C03633=1093.547,92.703,-61.297,175.902,17.512,152.547
C03634=1093.553,92.952,-61.315,175.903,17.513,152.547
C03635=1093.558,93.202,-61.333,175.906,17.514,152.547
C03636=1093.564,93.452,-61.351,175.908,17.515,152.547
C03637=1093.569,93.701,-61.369,175.911,17.516,152.546
C03638=1093.575,93.950,-61.386,175.913,17.517,152.546
C03639=1093.581,94.199,-61.405,175.915,17.518,152.546
C03640=1093.586,94.448,-61.423,175.918,17.519,152.546
C03641=1093.592,94.697,-61.441,175.920,17.520,152.545
C03642=1093.598,94.947,-61.459,175.923,17.521,152.545
C03643=1093.603,95.196,-61.476,175.925,17.522,152.545
C03644=1093.609,95.472,-61.497,175.927,17.523,152.545
C03645=1093.616,95.748,-61.516,175.930,17.524,152.544
C03646=1093.622,96.023,-61.536,175.933,17.525,152.544
C03647=1093.628,96.299,-61.557,175.935,17.526,152.544
C03648=1093.634,96.548,-61.575,175.938,17.528,152.544
C03649=1093.639,96.797,-61.592,175.940,17.529,152.543
C03650=1093.645,97.048,-61.611,175.942,17.530,152.543
C03651=1093.651,97.296,-61.629,175.944,17.531,152.543
C03652=1093.657,97.546,-61.647,175.947,17.532,152.543
C03653=1093.662,97.795,-61.664,175.950,17.533,152.542
C03654=1093.668,98.045,-61.683,175.952,17.534,152.542
C03655=1093.673,98.293,-61.701,175.954,17.535,152.542
C03656=1093.680,98.543,-61.719,175.956,17.535,152.542
C03657=1093.684,98.792,-61.737,175.959,17.537,152.541
C03658=1093.691,99.041,-61.756,175.961,17.537,152.541
C03659=1093.696,99.290,-61.773,175.964,17.538,152.541
C03660=1093.702,99.540,-61.791,175.966,17.540,152.541
C03661=1093.707,99.789,-61.810,175.968,17.540,152.540
C03662=1093.714,100.039,-61.828,175.971,17.541,152.540
C03663=1093.719,100.288,-61.846,175.973,17.542,152.540
C03664=1093.725,100.537,-61.865,175.976,17.543,152.540
C03665=1093.730,100.786,-61.883,175.978,17.545,152.539
C03666=1093.736,101.036,-61.901,175.980,17.545,152.539
C03667=1093.742,101.285,-61.919,175.983,17.546,152.539
C03668=1093.748,101.534,-61.937,175.985,17.547,152.538
C03669=1093.753,101.783,-61.956,175.988,17.548,152.538
C03670=1093.759,102.033,-61.974,175.990,17.549,152.538
C03671=1093.764,102.282,-61.993,175.992,17.550,152.538
C03672=1093.770,102.531,-62.011,175.995,17.551,152.537
C03673=1093.775,102.781,-62.029,175.998,17.552,152.537
C03674=1093.781,103.030,-62.048,176.000,17.553,152.537
C03675=1093.786,103.279,-62.066,176.002,17.554,152.537
C03676=1093.792,103.528,-62.085,176.004,17.555,152.536
C03677=1093.797,103.778,-62.103,176.007,17.556,152.536
C03678=1093.804,104.027,-62.121,176.010,17.557,152.536
C03679=1093.808,104.276,-62.140,176.012,17.558,152.536
C03680=1093.815,104.525,-62.158,176.014,17.559,152.535
C03681=1093.820,104.775,-62.176,176.016,17.559,152.535
C03682=1093.826,105.024,-62.195,176.019,17.560,152.535
C03683=1093.831,105.273,-62.213,176.022,17.562,152.534
C03684=1093.837,105.522,-62.232,176.024,17.562,152.534
C03685=1093.842,105.771,-62.251,176.027,17.563,152.534
C03686=1093.848,106.021,-62.269,176.029,17.565,152.534
C03687=1093.854,106.269,-62.288,176.031,17.565,152.533
C03688=1093.859,106.519,-62.306,176.034,17.566,152.533
C03689=1093.865,106.769,-62.325,176.036,17.567,152.533
C03690=1093.870,107.017,-62.344,176.039,17.568,152.532
C03691=1093.877,107.267,-62.362,176.041,17.569,152.532
C03692=1093.882,107.516,-62.380,176.043,17.570,152.532
C03693=1093.887,107.766,-62.399,176.046,17.571,152.532
C03694=1093.893,108.015,-62.418,176.049,17.572,152.531
C03695=1093.899,108.264,-62.436,176.051,17.573,152.531
C03696=1093.905,108.513,-62.454,176.054,17.573,152.531
C03697=1093.910,108.762,-62.473,176.056,17.574,152.530
C03698=1093.915,109.012,-62.492,176.058,17.575,152.530
C03699=1093.922,109.261,-62.510,176.061,17.576,152.530
C03700=1093.927,109.510,-62.529,176.063,17.577,152.530
C03701=1093.933,109.759,-62.548,176.066,17.578,152.529
C03702=1093.939,110.009,-62.567,176.069,17.579,152.529
C03703=1093.944,110.258,-62.585,176.071,17.580,152.529
C03704=1093.950,110.507,-62.604,176.073,17.581,152.528
C03705=1093.956,110.757,-62.623,176.075,17.581,152.528
C03706=1093.962,111.005,-62.642,176.078,17.582,152.528
C03707=1093.967,111.255,-62.660,176.081,17.583,152.528
C03708=1093.973,111.531,-62.681,176.084,17.584,152.527
C03709=1093.979,111.806,-62.702,176.087,17.585,152.527
C03710=1093.985,112.082,-62.723,176.089,17.586,152.527
C03711=1093.992,112.359,-62.744,176.092,17.587,152.526
C03712=1093.997,112.607,-62.762,176.094,17.588,152.526
C03713=1094.003,112.856,-62.781,176.097,17.589,152.526
C03714=1094.009,113.106,-62.801,176.099,17.589,152.525
C03715=1094.014,113.355,-62.819,176.102,17.590,152.525
C03716=1094.020,113.604,-62.837,176.105,17.592,152.525
C03717=1094.026,113.854,-62.857,176.107,17.592,152.524
C03718=1094.031,114.103,-62.876,176.109,17.593,152.524
C03719=1094.036,114.352,-62.895,176.112,17.594,152.524
C03720=1094.043,114.601,-62.913,176.114,17.595,152.524
C03721=1094.049,114.850,-62.933,176.117,17.595,152.523
C03722=1094.054,115.099,-62.952,176.120,17.597,152.523
C03723=1094.059,115.349,-62.971,176.122,17.597,152.523
C03724=1094.065,115.598,-62.990,176.124,17.598,152.522
C03725=1094.070,115.847,-63.009,176.127,17.599,152.522
C03726=1094.076,116.096,-63.028,176.129,17.600,152.522
C03727=1094.081,116.346,-63.047,176.132,17.601,152.521
C03728=1094.086,116.595,-63.066,176.134,17.602,152.521
C03729=1094.092,116.844,-63.085,176.137,17.602,152.521
C03730=1094.098,117.094,-63.104,176.140,17.604,152.520
C03731=1094.103,117.343,-63.123,176.142,17.604,152.520
C03732=1094.108,117.592,-63.142,176.145,17.605,152.520
C03733=1094.114,117.842,-63.161,176.147,17.606,152.520
C03734=1094.119,118.090,-63.180,176.149,17.607,152.519
C03735=1094.126,118.339,-63.199,176.152,17.607,152.519
C03736=1094.132,118.588,-63.219,176.155,17.609,152.519
C03737=1094.137,118.838,-63.238,176.157,17.609,152.518
C03738=1094.142,119.086,-63.257,176.160,17.610,152.518
C03739=1094.148,119.336,-63.276,176.163,17.611,152.518
C03740=1094.154,119.585,-63.295,176.165,17.611,152.517
C03741=1094.159,119.835,-63.315,176.167,17.613,152.517
C03742=1094.165,120.083,-63.334,176.170,17.614,152.517
C03743=1094.170,120.333,-63.353,176.172,17.614,152.516
C03744=1094.176,120.582,-63.372,176.175,17.615,152.516
C03745=1094.182,120.832,-63.391,176.178,17.616,152.516
C03746=1094.187,121.080,-63.410,176.181,17.617,152.515
C03747=1094.193,121.329,-63.430,176.183,17.617,152.515
C03748=1094.198,121.579,-63.449,176.186,17.618,152.515
C03749=1094.204,121.828,-63.469,176.188,17.620,152.515
C03750=1094.210,122.078,-63.488,176.191,17.620,152.514
C03751=1094.215,122.326,-63.507,176.193,17.621,152.514
C03752=1094.220,122.575,-63.527,176.196,17.622,152.513
C03753=1094.226,122.825,-63.547,176.198,17.622,152.513
C03754=1094.231,123.074,-63.566,176.201,17.623,152.513
C03755=1094.237,123.324,-63.585,176.204,17.624,152.512
C03756=1094.242,123.572,-63.604,176.206,17.624,152.512
C03757=1094.248,123.821,-63.624,176.209,17.626,152.512
C03758=1094.254,124.071,-63.643,176.212,17.626,152.511
C03759=1094.260,124.320,-63.662,176.214,17.627,152.511
C03760=1094.266,124.569,-63.682,176.217,17.628,152.511
C03761=1094.271,124.818,-63.702,176.220,17.628,152.510
C03762=1094.277,125.068,-63.721,176.222,17.629,152.510
C03763=1094.282,125.316,-63.740,176.225,17.630,152.510
C03764=1094.288,125.565,-63.760,176.227,17.631,152.509
C03765=1094.294,125.815,-63.779,176.229,17.631,152.509
C03766=1094.299,126.064,-63.798,176.232,17.632,152.509
C03767=1094.305,126.313,-63.819,176.235,17.633,152.508
C03768=1094.310,126.563,-63.838,176.238,17.634,152.508
C03769=1094.316,126.812,-63.858,176.240,17.634,152.508
C03770=1094.322,127.061,-63.877,176.243,17.635,152.507
C03771=1094.328,127.310,-63.896,176.246,17.636,152.507
C03772=1094.334,127.586,-63.918,176.249,17.637,152.506
C03773=1094.340,127.862,-63.940,176.252,17.638,152.506
C03774=1094.347,128.138,-63.961,176.255,17.639,152.506
C03775=1094.353,128.413,-63.983,176.258,17.639,152.505
C03776=1094.358,128.663,-64.003,176.260,17.639,152.505
C03777=1094.364,128.912,-64.023,176.263,17.641,152.505
C03778=1094.370,129.161,-64.042,176.266,17.641,152.504
C03779=1094.376,129.410,-64.062,176.268,17.642,152.504
C03780=1094.382,129.659,-64.081,176.271,17.642,152.503
C03781=1094.388,129.908,-64.101,176.274,17.643,152.503
C03782=1094.393,130.158,-64.121,176.276,17.644,152.503
C03783=1094.398,130.407,-64.141,176.279,17.644,152.502
C03784=1094.404,130.656,-64.160,176.282,17.645,152.502
C03785=1094.410,130.905,-64.180,176.284,17.646,152.502
C03786=1094.416,131.154,-64.200,176.287,17.646,152.501
C03787=1094.422,131.403,-64.220,176.290,17.647,152.501
C03788=1094.427,131.653,-64.239,176.293,17.648,152.500
C03789=1094.433,131.902,-64.259,176.294,17.649,152.500
C03790=1094.439,132.151,-64.279,176.297,17.649,152.500
C03791=1094.444,132.400,-64.299,176.300,17.650,152.499
C03792=1094.450,132.649,-64.319,176.303,17.650,152.499
C03793=1094.455,132.898,-64.338,176.305,17.651,152.499
C03794=1094.461,133.147,-64.358,176.308,17.652,152.498
C03795=1094.466,133.396,-64.379,176.311,17.653,152.498
C03796=1094.472,133.645,-64.398,176.313,17.653,152.498
C03797=1094.477,133.894,-64.418,176.316,17.654,152.497
C03798=1094.483,134.144,-64.438,176.319,17.655,152.497
C03799=1094.489,134.393,-64.458,176.322,17.656,152.496
C03800=1094.494,134.642,-64.478,176.324,17.656,152.496
C03801=1094.500,134.891,-64.498,176.327,17.657,152.496
C03802=1094.505,135.140,-64.518,176.330,17.658,152.495
C03803=1094.511,135.389,-64.538,176.332,17.658,152.495
C03804=1094.517,135.638,-64.558,176.335,17.659,152.495
C03805=1094.522,135.888,-64.578,176.338,17.659,152.494
C03806=1094.528,136.137,-64.598,176.341,17.661,152.494
C03807=1094.534,136.386,-64.619,176.343,17.661,152.493
C03808=1094.540,136.635,-64.638,176.346,17.661,152.493
C03809=1094.545,136.885,-64.658,176.349,17.662,152.493
C03810=1094.551,137.134,-64.678,176.352,17.663,152.492
C03811=1094.557,137.383,-64.698,176.354,17.663,152.492
C03812=1094.562,137.632,-64.719,176.357,17.664,152.492
C03813=1094.568,137.880,-64.739,176.360,17.665,152.491
C03814=1094.573,138.130,-64.759,176.362,17.665,152.491
C03815=1094.579,138.379,-64.779,176.365,17.666,152.490
C03816=1094.584,138.628,-64.799,176.368,17.667,152.490
C03817=1094.590,138.877,-64.819,176.371,17.667,152.490
C03818=1094.595,139.126,-64.840,176.373,17.668,152.489
C03819=1094.601,139.375,-64.860,176.376,17.668,152.489
C03820=1094.606,139.625,-64.879,176.379,17.669,152.488
C03821=1094.613,139.874,-64.900,176.382,17.670,152.488
C03822=1094.618,140.123,-64.920,176.384,17.670,152.488
C03823=1094.624,140.372,-64.940,176.387,17.671,152.487
C03824=1094.629,140.621,-64.961,176.390,17.672,152.487
C03825=1094.635,140.870,-64.981,176.393,17.673,152.486
C03826=1094.641,141.119,-65.001,176.395,17.673,152.486
C03827=1094.646,141.368,-65.022,176.398,17.674,152.486
C03828=1094.652,141.617,-65.042,176.401,17.674,152.485
C03829=1094.657,141.866,-65.062,176.404,17.675,152.485
C03830=1094.662,142.115,-65.083,176.406,17.675,152.484
C03831=1094.669,142.365,-65.103,176.409,17.676,152.484
C03832=1094.674,142.614,-65.124,176.412,17.677,152.484
C03833=1094.679,142.863,-65.144,176.415,17.677,152.483
C03834=1094.685,143.112,-65.164,176.418,17.678,152.483
C03835=1094.691,143.361,-65.185,176.420,17.679,152.482
C03836=1094.697,143.637,-65.207,176.424,17.679,152.482
C03837=1094.703,143.913,-65.230,176.427,17.680,152.482
C03838=1094.709,144.189,-65.253,176.430,17.681,152.481
C03839=1094.715,144.464,-65.275,176.432,17.681,152.481
C03840=1094.721,144.713,-65.295,176.435,17.682,152.480
C03841=1094.726,144.962,-65.316,176.438,17.683,152.480
C03842=1094.732,145.212,-65.337,176.441,17.683,152.479
C03843=1094.739,145.460,-65.357,176.444,17.684,152.479
C03844=1094.744,145.709,-65.378,176.447,17.684,152.479
C03845=1094.749,145.958,-65.399,176.450,17.685,152.478
C03846=1094.754,146.208,-65.419,176.453,17.685,152.478
C03847=1094.761,146.457,-65.439,176.455,17.686,152.477
C03848=1094.766,146.706,-65.460,176.458,17.686,152.477
C03849=1094.771,146.955,-65.481,176.461,17.687,152.476
C03850=1094.778,147.203,-65.501,176.464,17.688,152.476
C03851=1094.784,147.453,-65.522,176.467,17.689,152.476
C03852=1094.789,147.702,-65.543,176.469,17.689,152.475
C03853=1094.794,147.952,-65.563,176.472,17.689,152.475
C03854=1094.800,148.200,-65.583,176.475,17.690,152.474
C03855=1094.806,148.449,-65.604,176.478,17.690,152.474
C03856=1094.812,148.699,-65.625,176.481,17.691,152.473
C03857=1094.817,148.948,-65.646,176.484,17.691,152.473
C03858=1094.822,149.197,-65.666,176.487,17.692,152.473
C03859=1094.828,149.445,-65.688,176.490,17.693,152.472
C03860=1094.834,149.695,-65.708,176.493,17.694,152.472
C03861=1094.839,149.944,-65.729,176.495,17.694,152.471
C03862=1094.845,150.193,-65.750,176.498,17.694,152.471
C03863=1094.850,150.442,-65.770,176.501,17.695,152.471
C03864=1094.856,150.692,-65.791,176.504,17.695,152.470
C03865=1094.862,150.940,-65.813,176.506,17.696,152.470
C03866=1094.867,151.189,-65.833,176.509,17.696,152.469
C03867=1094.872,151.438,-65.854,176.512,17.697,152.469
C03868=1094.878,151.687,-65.875,176.515,17.698,152.468
C03869=1094.884,151.936,-65.895,176.518,17.699,152.468
C03870=1094.890,152.185,-65.916,176.520,17.698,152.467
C03871=1094.896,152.435,-65.938,176.523,17.699,152.467
C03872=1094.901,152.684,-65.958,176.526,17.700,152.467
C03873=1094.907,152.932,-65.979,176.529,17.701,152.466
C03874=1094.912,153.181,-66.000,176.532,17.701,152.466
C03875=1094.918,153.431,-66.021,176.535,17.701,152.465
C03876=1094.923,153.680,-66.042,176.538,17.702,152.465
C03877=1094.929,153.929,-66.063,176.541,17.702,152.464
C03878=1094.935,154.178,-66.084,176.544,17.703,152.464
C03879=1094.940,154.427,-66.105,176.547,17.704,152.463
C03880=1094.946,154.676,-66.126,176.549,17.704,152.463
C03881=1094.951,154.925,-66.147,176.552,17.704,152.463
C03882=1094.957,155.174,-66.168,176.555,17.705,152.462
C03883=1094.962,155.423,-66.189,176.559,17.705,152.462
C03884=1094.968,155.672,-66.210,176.561,17.706,152.461
C03885=1094.974,155.921,-66.231,176.564,17.706,152.461
C03886=1094.979,156.170,-66.252,176.567,17.707,152.460
C03887=1094.985,156.420,-66.273,176.570,17.707,152.460
C03888=1094.991,156.668,-66.294,176.573,17.708,152.460
C03889=1094.997,156.917,-66.316,176.576,17.709,152.459
C03890=1095.002,157.167,-66.337,176.578,17.709,152.459
C03891=1095.008,157.415,-66.358,176.581,17.709,152.458
C03892=1095.013,157.665,-66.379,176.584,17.710,152.458
C03893=1095.018,157.914,-66.401,176.587,17.711,152.457
C03894=1095.024,158.162,-66.422,176.591,17.711,152.457
C03895=1095.030,158.412,-66.443,176.594,17.712,152.456
C03896=1095.035,158.661,-66.464,176.596,17.712,152.456
C03897=1095.041,158.910,-66.486,176.599,17.712,152.455
C03898=1095.047,159.159,-66.506,176.602,17.713,152.455
C03899=1095.052,159.407,-66.528,176.605,17.714,152.455
C03900=1095.058,159.683,-66.552,176.608,17.714,152.454
C03901=1095.065,159.958,-66.575,176.611,17.714,152.453
C03902=1095.071,160.234,-66.599,176.614,17.715,152.453
C03903=1095.077,160.509,-66.622,176.618,17.715,152.453
C03904=1095.083,160.759,-66.643,176.621,17.716,152.452
C03905=1095.088,161.008,-66.665,176.624,17.716,152.452
C03906=1095.094,161.256,-66.686,176.627,17.717,152.451
C03907=1095.099,161.506,-66.708,176.630,17.717,152.451
C03908=1095.105,161.754,-66.729,176.632,17.718,152.450
C03909=1095.111,162.004,-66.750,176.635,17.718,152.450
C03910=1095.116,162.253,-66.772,176.639,17.719,152.449
C03911=1095.121,162.501,-66.793,176.642,17.719,152.449
C03912=1095.127,162.751,-66.815,176.645,17.720,152.448
C03913=1095.132,162.999,-66.837,176.648,17.720,152.448
C03914=1095.138,163.249,-66.858,176.651,17.721,152.447
C03915=1095.143,163.498,-66.880,176.653,17.721,152.447
C03916=1095.149,163.747,-66.901,176.656,17.722,152.446
C03917=1095.155,163.996,-66.923,176.659,17.722,152.446
C03918=1095.159,164.245,-66.945,176.662,17.723,152.446
C03919=1095.166,164.494,-66.966,176.665,17.723,152.445
C03920=1095.170,164.743,-66.988,176.668,17.724,152.445
C03921=1095.176,164.992,-67.009,176.671,17.724,152.444
C03922=1095.181,165.241,-67.031,176.674,17.725,152.444
C03923=1095.187,165.490,-67.052,176.677,17.725,152.443
C03924=1095.193,165.739,-67.074,176.680,17.726,152.443
C03925=1095.198,165.988,-67.096,176.683,17.726,152.442
C03926=1095.204,166.237,-67.117,176.686,17.727,152.442
C03927=1095.209,166.486,-67.139,176.689,17.728,152.441
C03928=1095.215,166.735,-67.161,176.691,17.728,152.441
C03929=1095.220,166.984,-67.183,176.695,17.728,152.440
C03930=1095.226,167.233,-67.204,176.698,17.729,152.440
C03931=1095.231,167.482,-67.226,176.701,17.729,152.439
C03932=1095.237,167.731,-67.248,176.704,17.730,152.439
C03933=1095.242,167.980,-67.270,176.707,17.730,152.439
C03934=1095.248,168.229,-67.291,176.710,17.731,152.438
C03935=1095.253,168.478,-67.313,176.713,17.731,152.438
C03936=1095.259,168.727,-67.335,176.716,17.731,152.437
C03937=1095.264,168.975,-67.357,176.719,17.732,152.437
C03938=1095.270,169.224,-67.379,176.722,17.732,152.436
C03939=1095.276,169.474,-67.401,176.725,17.733,152.436
C03940=1095.281,169.723,-67.422,176.728,17.733,152.435
C03941=1095.287,169.972,-67.445,176.731,17.734,152.435
C03942=1095.292,170.221,-67.466,176.734,17.734,152.434
C03943=1095.297,170.470,-67.488,176.737,17.734,152.434
C03944=1095.303,170.719,-67.509,176.740,17.735,152.433
C03945=1095.309,170.967,-67.532,176.743,17.735,152.433
C03946=1095.315,171.217,-67.554,176.746,17.735,152.432
C03947=1095.320,171.465,-67.576,176.749,17.736,152.432
C03948=1095.326,171.715,-67.598,176.752,17.737,152.431
C03949=1095.331,171.963,-67.619,176.755,17.737,152.431
C03950=1095.336,172.212,-67.642,176.759,17.738,152.430
C03951=1095.343,172.462,-67.664,176.761,17.737,152.430
C03952=1095.347,172.710,-67.686,176.764,17.738,152.429
C03953=1095.354,172.960,-67.707,176.767,17.738,152.429
C03954=1095.359,173.208,-67.730,176.770,17.739,152.428
C03955=1095.365,173.457,-67.752,176.774,17.739,152.428
C03956=1095.370,173.707,-67.774,176.777,17.740,152.427
C03957=1095.375,173.955,-67.796,176.780,17.740,152.427
C03958=1095.382,174.204,-67.818,176.783,17.741,152.426
C03959=1095.387,174.453,-67.840,176.786,17.740,152.426
C03960=1095.393,174.702,-67.862,176.789,17.741,152.425
C03961=1095.398,174.951,-67.885,176.792,17.742,152.425
C03962=1095.404,175.200,-67.907,176.795,17.742,152.424
C03963=1095.410,175.448,-67.929,176.798,17.742,152.424
C03964=1095.416,175.724,-67.953,176.802,17.742,152.423
C03965=1095.422,175.999,-67.978,176.805,17.743,152.423
C03966=1095.428,176.274,-68.002,176.809,17.744,152.422
C03967=1095.434,176.549,-68.027,176.812,17.744,152.421
C03968=1095.440,176.798,-68.049,176.815,17.745,152.421
C03969=1095.446,177.047,-68.072,176.818,17.745,152.420
C03970=1095.451,177.297,-68.094,176.822,17.745,152.420
C03971=1095.457,177.544,-68.116,176.824,17.745,152.419
C03972=1095.463,177.794,-68.138,176.827,17.745,152.419
C03973=1095.468,178.043,-68.161,176.830,17.746,152.418
C03974=1095.474,178.292,-68.183,176.834,17.746,152.418
C03975=1095.480,178.540,-68.205,176.837,17.747,152.417
C03976=1095.485,178.790,-68.227,176.840,17.747,152.417
C03977=1095.491,179.038,-68.250,176.843,17.747,152.416
C03978=1095.497,179.288,-68.272,176.846,17.748,152.416
C03979=1095.503,179.537,-68.295,176.850,17.748,152.415
C03980=1095.508,179.785,-68.316,176.853,17.749,152.415
C03981=1095.514,180.034,-68.339,176.855,17.748,152.414
C03982=1095.520,180.283,-68.362,176.858,17.749,152.414
C03983=1095.525,180.533,-68.384,176.862,17.749,152.413
C03984=1095.532,180.781,-68.407,176.865,17.749,152.412
C03985=1095.536,181.030,-68.429,176.868,17.750,152.412
C03986=1095.542,181.279,-68.451,176.871,17.750,152.412
C03987=1095.548,181.528,-68.474,176.874,17.751,152.411
C03988=1095.554,181.777,-68.496,176.878,17.751,152.410
C03989=1095.560,182.026,-68.519,176.881,17.751,152.410
C03990=1095.565,182.275,-68.542,176.884,17.751,152.409
C03991=1095.570,182.524,-68.564,176.887,17.752,152.409
C03992=1095.577,182.772,-68.586,176.891,17.752,152.408
C03993=1095.582,183.021,-68.609,176.893,17.752,152.408
C03994=1095.588,183.271,-68.631,176.896,17.752,152.407
C03995=1095.594,183.520,-68.654,176.900,17.752,152.407
C03996=1095.600,183.768,-68.677,176.903,17.753,152.406
C03997=1095.606,184.017,-68.700,176.906,17.753,152.405
C03998=1095.611,184.267,-68.722,176.909,17.753,152.405
C03999=1095.617,184.515,-68.745,176.913,17.754,152.404
C04000=1095.622,184.764,-68.767,176.916,17.754,152.404
C04001=1095.629,185.012,-68.790,176.919,17.754,152.403
C04002=1095.634,185.261,-68.813,176.922,17.755,152.403
C04003=1095.640,185.511,-68.835,176.925,17.755,152.402
C04004=1095.645,185.760,-68.858,176.929,17.756,152.402
C04005=1095.650,186.009,-68.881,176.932,17.756,152.401
C04006=1095.656,186.257,-68.904,176.935,17.756,152.401
C04007=1095.661,186.506,-68.927,176.938,17.757,152.400
C04008=1095.667,186.755,-68.950,176.941,17.757,152.400
C04009=1095.672,187.004,-68.972,176.944,17.757,152.399
C04010=1095.678,187.253,-68.995,176.947,17.757,152.399
C04011=1095.684,187.502,-69.018,176.950,17.758,152.398
C04012=1095.689,187.750,-69.040,176.954,17.758,152.397
C04013=1095.694,187.999,-69.064,176.957,17.758,152.397
C04014=1095.700,188.248,-69.087,176.960,17.759,152.396
C04015=1095.706,188.497,-69.110,176.963,17.759,152.396
C04016=1095.711,188.746,-69.133,176.966,17.760,152.395
C04017=1095.717,188.995,-69.156,176.970,17.760,152.395
C04018=1095.723,189.244,-69.179,176.973,17.760,152.394
C04019=1095.728,189.492,-69.201,176.976,17.761,152.394
C04020=1095.733,189.741,-69.225,176.979,17.761,152.393
C04021=1095.739,189.990,-69.248,176.983,17.761,152.393
C04022=1095.744,190.239,-69.271,176.986,17.762,152.392
C04023=1095.750,190.488,-69.294,176.989,17.762,152.392
C04024=1095.756,190.737,-69.317,176.992,17.762,152.391
C04025=1095.761,190.986,-69.340,176.996,17.763,152.390
C04026=1095.766,191.235,-69.363,176.999,17.763,152.390
C04027=1095.772,191.484,-69.386,177.002,17.763,152.389
C04028=1095.778,191.758,-69.411,177.005,17.763,152.389
C04029=1095.784,192.034,-69.437,177.009,17.764,152.388
C04030=1095.791,192.308,-69.462,177.013,17.765,152.388
C04031=1095.796,192.583,-69.488,177.016,17.765,152.387
C04032=1095.802,192.832,-69.511,177.019,17.765,152.386
C04033=1095.808,193.081,-69.534,177.023,17.765,152.386
C04034=1095.813,193.329,-69.557,177.026,17.765,152.385
C04035=1095.819,193.578,-69.581,177.029,17.766,152.385
C04036=1095.824,193.827,-69.604,177.032,17.766,152.384
C04037=1095.830,194.076,-69.627,177.036,17.766,152.384
C04038=1095.836,194.325,-69.650,177.039,17.767,152.383
C04039=1095.842,194.574,-69.673,177.042,17.767,152.382
C04040=1095.847,194.822,-69.697,177.045,17.767,152.382
C04041=1095.853,195.071,-69.720,177.049,17.768,152.381
C04042=1095.858,195.320,-69.743,177.052,17.768,152.381
C04043=1095.863,195.569,-69.767,177.055,17.768,152.380
C04044=1095.869,195.818,-69.791,177.058,17.769,152.380
C04045=1095.875,196.066,-69.813,177.062,17.769,152.379
C04046=1095.881,196.315,-69.836,177.065,17.769,152.378
C04047=1095.886,196.564,-69.861,177.068,17.769,152.378
C04048=1095.892,196.813,-69.884,177.072,17.769,152.377
C04049=1095.898,197.062,-69.907,177.075,17.770,152.377
C04050=1095.904,197.311,-69.931,177.078,17.770,152.376
C04051=1095.909,197.560,-69.954,177.081,17.770,152.376
C04052=1095.915,197.809,-69.977,177.085,17.771,152.375
C04053=1095.920,198.057,-70.001,177.088,17.771,152.375
C04054=1095.926,198.306,-70.024,177.091,17.771,152.374
C04055=1095.932,198.555,-70.047,177.095,17.771,152.373
C04056=1095.937,198.804,-70.072,177.098,17.772,152.373
C04057=1095.943,199.053,-70.094,177.101,17.772,152.372
C04058=1095.949,199.301,-70.118,177.104,17.772,152.372
C04059=1095.954,199.550,-70.142,177.108,17.772,152.371
C04060=1095.960,199.799,-70.166,177.111,17.772,152.370
C04061=1095.965,200.048,-70.189,177.114,17.773,152.370
C04062=1095.972,200.297,-70.213,177.118,17.773,152.369
C04063=1095.977,200.545,-70.236,177.121,17.773,152.369
C04064=1095.983,200.794,-70.260,177.124,17.773,152.368
C04065=1095.988,201.043,-70.283,177.128,17.774,152.368
C04066=1095.995,201.292,-70.307,177.131,17.774,152.367
C04067=1096.000,201.541,-70.331,177.134,17.774,152.366
C04068=1096.006,201.789,-70.354,177.138,17.774,152.366
C04069=1096.011,202.039,-70.378,177.141,17.774,152.365
C04070=1096.017,202.287,-70.401,177.144,17.775,152.365
C04071=1096.023,202.537,-70.425,177.147,17.775,152.364
C04072=1096.029,202.785,-70.449,177.151,17.775,152.363
C04073=1096.034,203.034,-70.473,177.154,17.775,152.363
C04074=1096.040,203.283,-70.496,177.157,17.776,152.362
C04075=1096.045,203.531,-70.520,177.161,17.776,152.362
C04076=1096.051,203.780,-70.543,177.164,17.776,152.361
C04077=1096.057,204.029,-70.568,177.167,17.777,152.361
C04078=1096.063,204.278,-70.592,177.171,17.776,152.360
C04079=1096.068,204.527,-70.615,177.174,17.777,152.359
C04080=1096.073,204.775,-70.640,177.177,17.777,152.359
C04081=1096.079,205.024,-70.663,177.180,17.777,152.358
C04082=1096.084,205.273,-70.687,177.184,17.778,152.358
C04083=1096.090,205.522,-70.711,177.187,17.778,152.357
C04084=1096.096,205.770,-70.735,177.190,17.778,152.357
C04085=1096.101,206.019,-70.759,177.194,17.778,152.356
C04086=1096.106,206.268,-70.783,177.197,17.779,152.355
C04087=1096.112,206.517,-70.806,177.200,17.779,152.355
C04088=1096.118,206.766,-70.831,177.204,17.779,152.354
C04089=1096.123,207.014,-70.855,177.207,17.779,152.354
C04090=1096.129,207.263,-70.879,177.211,17.780,152.353
C04091=1096.134,207.512,-70.903,177.214,17.780,152.353
C04092=1096.158,208.525,-71.001,177.264,17.800,152.347
C04093=1096.166,208.898,-71.037,177.269,17.802,152.347
C04094=1096.175,209.271,-71.073,177.274,17.804,152.346
C04095=1096.183,209.644,-71.111,177.279,17.805,152.346
C04096=1096.192,210.017,-71.147,177.283,17.807,152.345
C04097=1096.197,210.265,-71.172,177.286,17.808,152.345
C04098=1096.202,210.514,-71.196,177.290,17.809,152.344
C04099=1096.208,210.763,-71.220,177.293,17.810,152.344
C04100=1096.214,211.012,-71.245,177.296,17.811,152.344
C04101=1096.220,211.260,-71.268,177.300,17.813,152.343
C04102=1096.226,211.509,-71.293,177.302,17.814,152.343
C04103=1096.231,211.758,-71.317,177.305,17.814,152.343
C04104=1096.237,212.007,-71.342,177.309,17.816,152.342
C04105=1096.242,212.255,-71.367,177.312,17.817,152.342
C04106=1096.248,212.504,-71.391,177.316,17.818,152.341
C04107=1096.254,212.753,-71.416,177.319,17.819,152.341
C04108=1096.259,213.002,-71.440,177.321,17.821,152.341
C04109=1096.265,213.251,-71.465,177.325,17.822,152.340
C04110=1096.270,213.499,-71.490,177.328,17.823,152.340
C04111=1096.276,213.748,-71.514,177.331,17.824,152.340
C04112=1096.282,213.997,-71.538,177.335,17.825,152.339
C04113=1096.287,214.245,-71.563,177.338,17.826,152.339
C04114=1096.292,214.494,-71.589,177.341,17.827,152.339
C04115=1096.298,214.743,-71.613,177.344,17.829,152.338
C04116=1096.304,214.992,-71.637,177.347,17.830,152.338
C04117=1096.309,215.240,-71.662,177.351,17.831,152.338
C04118=1096.314,215.489,-71.687,177.354,17.832,152.337
C04119=1096.320,215.738,-71.711,177.356,17.833,152.337
C04120=1096.326,215.986,-71.736,177.360,17.834,152.337
C04121=1096.332,216.235,-71.761,177.363,17.836,152.336
C04122=1096.337,216.484,-71.786,177.366,17.836,152.336
C04123=1096.343,216.733,-71.811,177.370,17.838,152.335
C04124=1096.348,216.982,-71.835,177.373,17.839,152.335
C04125=1096.354,217.230,-71.861,177.376,17.841,152.335
C04126=1096.359,217.479,-71.885,177.379,17.841,152.334
C04127=1096.366,217.727,-71.910,177.382,17.842,152.334
C04128=1096.371,217.976,-71.935,177.386,17.844,152.334
C04129=1096.376,218.225,-71.960,177.389,17.845,152.333
C04130=1096.382,218.474,-71.985,177.392,17.846,152.333
C04131=1096.388,218.722,-72.010,177.395,17.847,152.333
C04132=1096.393,218.971,-72.034,177.398,17.848,152.332
C04133=1096.399,219.220,-72.060,177.402,17.850,152.332
C04134=1096.404,219.468,-72.085,177.405,17.850,152.332
C04135=1096.410,219.717,-72.110,177.409,17.852,152.331
C04136=1096.415,219.966,-72.134,177.411,17.853,152.331
C04137=1096.422,220.214,-72.159,177.414,17.854,152.331
C04138=1096.427,220.464,-72.185,177.418,17.855,152.330
C04139=1096.432,220.712,-72.210,177.421,17.857,152.330
C04140=1096.439,220.961,-72.235,177.425,17.858,152.329
C04141=1096.444,221.209,-72.259,177.427,17.859,152.329
C04142=1096.450,221.458,-72.285,177.430,17.860,152.329
C04143=1096.455,221.707,-72.310,177.434,17.861,152.328
C04144=1096.461,221.955,-72.335,177.437,17.862,152.328
C04145=1096.470,222.332,-72.373,177.442,17.864,152.327
C04146=1096.478,222.709,-72.411,177.447,17.866,152.327
C04147=1096.487,223.086,-72.450,177.452,17.868,152.326
C04148=1096.495,223.463,-72.488,177.457,17.870,152.326
C04149=1096.500,223.711,-72.513,177.460,17.870,152.326
C04150=1096.506,223.959,-72.538,177.463,17.872,152.325
C04151=1096.512,224.208,-72.564,177.466,17.873,152.325
C04152=1096.517,224.457,-72.588,177.470,17.875,152.324
C04153=1096.523,224.706,-72.614,177.473,17.876,152.324
C04154=1096.529,224.954,-72.639,177.476,17.877,152.324
C04155=1096.534,225.203,-72.665,177.479,17.878,152.323
C04156=1096.540,225.451,-72.690,177.483,17.880,152.323
C04157=1096.545,225.701,-72.716,177.486,17.881,152.323
C04158=1096.551,225.949,-72.741,177.489,17.881,152.322
C04159=1096.556,226.198,-72.766,177.493,17.883,152.322
C04160=1096.562,226.446,-72.791,177.495,17.884,152.322
C04161=1096.568,226.695,-72.817,177.499,17.886,152.321
C04162=1096.573,226.944,-72.843,177.502,17.886,152.321
C04163=1096.580,227.192,-72.868,177.505,17.888,152.321
C04164=1096.584,227.441,-72.894,177.508,17.889,152.320
C04165=1096.591,227.689,-72.919,177.512,17.890,152.320
C04166=1096.596,227.938,-72.945,177.515,17.892,152.320
C04167=1096.601,228.186,-72.970,177.518,17.892,152.319
C04168=1096.607,228.435,-72.996,177.522,17.894,152.319
C04169=1096.613,228.684,-73.022,177.524,17.895,152.319
C04170=1096.619,228.933,-73.047,177.528,17.897,152.318
C04171=1096.624,229.181,-73.073,177.531,17.897,152.318
C04172=1096.630,229.430,-73.098,177.535,17.899,152.318
C04173=1096.635,229.679,-73.124,177.538,17.900,152.317
C04174=1096.642,229.927,-73.149,177.541,17.901,152.317
C04175=1096.647,230.176,-73.175,177.544,17.903,152.317
C04176=1096.653,230.424,-73.200,177.548,17.904,152.316
C04177=1096.658,230.673,-73.226,177.551,17.905,152.316
C04178=1096.664,230.922,-73.252,177.554,17.907,152.316
C04179=1096.669,231.170,-73.277,177.557,17.908,152.315
C04180=1096.675,231.419,-73.303,177.561,17.909,152.315
C04181=1096.680,231.668,-73.329,177.564,17.910,152.315
C04182=1096.686,231.917,-73.356,177.568,17.912,152.314
C04183=1096.692,232.165,-73.380,177.570,17.913,152.314
C04184=1096.697,232.414,-73.406,177.573,17.914,152.314
C04185=1096.703,232.663,-73.432,177.577,17.915,152.313
C04186=1096.709,232.911,-73.458,177.580,17.916,152.313
C04187=1096.715,233.160,-73.484,177.583,17.918,152.312
C04188=1096.719,233.408,-73.510,177.586,17.919,152.312
C04189=1096.725,233.657,-73.536,177.590,17.920,152.312
C04190=1096.731,233.905,-73.561,177.593,17.921,152.311
C04191=1096.737,234.154,-73.588,177.596,17.923,152.311
C04192=1096.742,234.403,-73.614,177.599,17.924,152.311
C04193=1096.748,234.652,-73.640,177.603,17.925,152.310
C04194=1096.753,234.900,-73.665,177.606,17.927,152.310
C04195=1096.759,235.148,-73.691,177.610,17.928,152.310
C04196=1096.765,235.397,-73.717,177.612,17.929,152.310
C04197=1096.773,235.765,-73.756,177.618,17.931,152.309
C04198=1096.781,236.133,-73.794,177.623,17.933,152.309
C04199=1096.790,236.501,-73.833,177.627,17.935,152.308
C04200=1096.798,236.869,-73.872,177.632,17.937,152.308
C04201=1096.803,237.118,-73.897,177.635,17.939,152.307
C04202=1096.809,237.366,-73.924,177.638,17.940,152.307
C04203=1096.814,237.615,-73.950,177.642,17.941,152.307
C04204=1096.820,237.864,-73.977,177.645,17.942,152.306
C04205=1096.826,238.113,-74.003,177.649,17.944,152.306
C04206=1096.831,238.361,-74.029,177.651,17.945,152.306
C04207=1096.837,238.610,-74.055,177.655,17.946,152.305
C04208=1096.843,238.858,-74.082,177.658,17.948,152.305
C04209=1096.848,239.107,-74.108,177.662,17.949,152.305
C04210=1096.854,239.356,-74.134,177.664,17.950,152.304
C04211=1096.860,239.604,-74.159,177.668,17.952,152.304
C04212=1096.865,239.852,-74.186,177.672,17.953,152.304
C04213=1096.871,240.101,-74.212,177.675,17.954,152.303
C04214=1096.877,240.349,-74.239,177.678,17.956,152.303
C04215=1096.882,240.598,-74.265,177.681,17.957,152.303
C04216=1096.888,240.847,-74.291,177.685,17.958,152.302
C04217=1096.894,241.095,-74.318,177.688,17.959,152.302
C04218=1096.899,241.344,-74.344,177.691,17.961,152.302
C04219=1096.905,241.592,-74.370,177.694,17.962,152.301
C04220=1096.911,241.841,-74.397,177.698,17.964,152.301
C04221=1096.916,242.090,-74.423,177.701,17.965,152.301
C04222=1096.922,242.338,-74.450,177.704,17.966,152.300
C04223=1096.928,242.586,-74.476,177.707,17.967,152.300
C04224=1096.933,242.835,-74.503,177.711,17.969,152.300
C04225=1096.939,243.084,-74.529,177.714,17.971,152.299
C04226=1096.944,243.332,-74.556,177.717,17.971,152.299
C04227=1096.950,243.581,-74.583,177.721,17.973,152.299
C04228=1096.955,243.829,-74.609,177.724,17.974,152.298
C04229=1096.961,244.078,-74.635,177.727,17.976,152.298
C04230=1096.967,244.326,-74.662,177.730,17.977,152.298
C04231=1096.972,244.575,-74.689,177.734,17.979,152.298
C04232=1096.977,244.824,-74.716,177.738,17.980,152.297
C04233=1096.983,245.072,-74.743,177.740,17.981,152.297
C04234=1096.989,245.321,-74.768,177.744,17.983,152.296
C04235=1096.994,245.569,-74.795,177.747,17.984,152.296
C04236=1097.000,245.818,-74.822,177.750,17.986,152.296
C04237=1097.005,246.066,-74.849,177.753,17.987,152.296
C04238=1097.011,246.315,-74.876,177.757,17.988,152.295
C04239=1097.017,246.563,-74.902,177.761,17.990,152.295
C04240=1097.023,246.811,-74.929,177.763,17.991,152.295
C04241=1097.028,247.060,-74.956,177.767,17.993,152.294
C04242=1097.034,247.309,-74.983,177.770,17.994,152.294
C04243=1097.040,247.557,-75.010,177.773,17.995,152.294
C04244=1097.046,247.806,-75.037,177.776,17.997,152.294
C04245=1097.051,248.054,-75.064,177.780,17.998,152.293
C04246=1097.056,248.303,-75.090,177.783,18.000,152.293
C04247=1097.061,248.551,-75.118,177.786,18.001,152.293
C04248=1097.067,248.800,-75.144,177.790,18.003,152.292
C04249=1097.075,249.161,-75.183,177.794,18.005,152.292
C04250=1097.083,249.522,-75.222,177.799,18.006,152.291
C04251=1097.091,249.884,-75.261,177.804,18.009,152.291
C04252=1097.099,250.245,-75.301,177.809,18.011,152.291
C04253=1097.105,250.493,-75.328,177.812,18.012,152.290
C04254=1097.110,250.742,-75.355,177.815,18.014,152.290
C04255=1097.116,250.990,-75.381,177.819,18.016,152.290
C04256=1097.122,251.238,-75.409,177.822,18.017,152.289
C04257=1097.127,251.487,-75.436,177.825,18.018,152.289
C04258=1097.133,251.736,-75.463,177.829,18.020,152.289
C04259=1097.138,251.985,-75.490,177.832,18.021,152.289
C04260=1097.144,252.233,-75.517,177.835,18.023,152.288
C04261=1097.149,252.481,-75.545,177.838,18.024,152.288
C04262=1097.155,252.729,-75.572,177.842,18.026,152.288
C04263=1097.160,252.978,-75.599,177.845,18.027,152.287
C04264=1097.166,253.227,-75.626,177.848,18.029,152.287
C04265=1097.172,253.475,-75.654,177.852,18.030,152.287
C04266=1097.177,253.723,-75.680,177.855,18.031,152.287
C04267=1097.182,253.972,-75.708,177.858,18.033,152.286
C04268=1097.189,254.220,-75.735,177.862,18.035,152.286
C04269=1097.194,254.469,-75.763,177.865,18.036,152.286
C04270=1097.200,254.718,-75.789,177.868,18.037,152.285
C04271=1097.205,254.966,-75.817,177.872,18.039,152.285
C04272=1097.211,255.214,-75.844,177.874,18.041,152.285
C04273=1097.217,255.463,-75.872,177.878,18.042,152.284
C04274=1097.222,255.711,-75.899,177.882,18.044,152.284
C04275=1097.228,255.960,-75.926,177.885,18.045,152.284
C04276=1097.233,256.208,-75.954,177.888,18.046,152.284
C04277=1097.240,256.457,-75.981,177.891,18.048,152.283
C04278=1097.245,256.706,-76.008,177.895,18.049,152.283
C04279=1097.251,256.953,-76.036,177.898,18.051,152.283
C04280=1097.256,257.202,-76.063,177.901,18.052,152.282
C04281=1097.262,257.451,-76.091,177.905,18.054,152.282
C04282=1097.267,257.699,-76.118,177.908,18.056,152.282
C04283=1097.273,257.947,-76.146,177.911,18.056,152.281
C04284=1097.279,258.196,-76.173,177.915,18.058,152.281
C04285=1097.284,258.444,-76.201,177.918,18.060,152.281
C04286=1097.290,258.692,-76.229,177.921,18.061,152.281
C04287=1097.296,258.941,-76.255,177.925,18.063,152.280
C04288=1097.302,259.189,-76.284,177.928,18.065,152.280
C04289=1097.307,259.438,-76.310,177.931,18.066,152.280
C04290=1097.313,259.686,-76.338,177.935,18.067,152.280
C04291=1097.319,259.935,-76.367,177.938,18.069,152.279
C04292=1097.324,260.183,-76.393,177.941,18.070,152.279
C04293=1097.330,260.432,-76.422,177.945,18.072,152.279
C04294=1097.336,260.680,-76.450,177.948,18.073,152.278
C04295=1097.341,260.928,-76.476,177.951,18.075,152.278
C04296=1097.347,261.177,-76.505,177.955,18.076,152.278
C04297=1097.353,261.425,-76.533,177.958,18.078,152.277
C04298=1097.358,261.673,-76.559,177.961,18.079,152.277
C04299=1097.364,261.922,-76.588,177.965,18.081,152.277
C04300=1097.370,262.170,-76.616,177.968,18.083,152.277
C04301=1097.378,262.529,-76.656,177.973,18.085,152.276
C04302=1097.387,262.887,-76.696,177.977,18.087,152.276
C04303=1097.395,263.245,-76.735,177.982,18.089,152.275
C04304=1097.404,263.603,-76.776,177.987,18.091,152.275
C04305=1097.409,263.852,-76.804,177.990,18.092,152.275
C04306=1097.414,264.100,-76.832,177.994,18.094,152.274
C04307=1097.421,264.349,-76.859,177.997,18.096,152.274
C04308=1097.427,264.597,-76.887,178.001,18.098,152.274
C04309=1097.432,264.845,-76.915,178.003,18.099,152.274
C04310=1097.438,265.094,-76.944,178.007,18.100,152.273
C04311=1097.443,265.342,-76.971,178.011,18.102,152.273
C04312=1097.449,265.591,-77.000,178.013,18.104,152.273
C04313=1097.454,265.839,-77.028,178.017,18.105,152.273
C04314=1097.460,266.087,-77.056,178.020,18.107,152.272
C04315=1097.466,266.335,-77.084,178.023,18.108,152.272
C04316=1097.471,266.583,-77.112,178.027,18.110,152.272
C04317=1097.477,266.832,-77.140,178.030,18.112,152.271
C04318=1097.482,267.080,-77.168,178.034,18.114,152.271
C04319=1097.488,267.329,-77.197,178.037,18.115,152.271
C04320=1097.494,267.577,-77.225,178.040,18.116,152.271
C04321=1097.500,267.826,-77.253,178.044,18.118,152.270
C04322=1097.505,268.074,-77.281,178.047,18.120,152.270
C04323=1097.511,268.323,-77.309,178.050,18.121,152.270
C04324=1097.516,268.571,-77.337,178.054,18.123,152.270
C04325=1097.522,268.819,-77.365,178.057,18.125,152.269
C04326=1097.527,269.067,-77.393,178.060,18.126,152.269
C04327=1097.533,269.316,-77.422,178.064,18.128,152.269
C04328=1097.539,269.564,-77.450,178.067,18.130,152.269
C04329=1097.545,269.812,-77.479,178.070,18.131,152.268
C04330=1097.550,270.060,-77.507,178.073,18.133,152.268
C04331=1097.556,270.309,-77.535,178.077,18.134,152.268
C04332=1097.562,270.557,-77.563,178.080,18.136,152.268
C04333=1097.568,270.806,-77.591,178.083,18.138,152.267
C04334=1097.572,271.054,-77.621,178.087,18.139,152.267
C04335=1097.578,271.303,-77.649,178.090,18.141,152.267
C04336=1097.584,271.551,-77.677,178.094,18.143,152.267
C04337=1097.590,271.799,-77.705,178.096,18.144,152.266
C04338=1097.595,272.047,-77.734,178.100,18.146,152.266
C04339=1097.601,272.295,-77.762,178.103,18.148,152.266
C04340=1097.607,272.544,-77.791,178.107,18.150,152.266
C04341=1097.612,272.792,-77.820,178.110,18.151,152.265
C04342=1097.618,273.041,-77.848,178.113,18.153,152.265
C04343=1097.623,273.289,-77.876,178.117,18.155,152.265
C04344=1097.630,273.537,-77.905,178.120,18.157,152.265
C04345=1097.636,273.786,-77.933,178.123,18.158,152.265
C04346=1097.641,274.033,-77.963,178.126,18.160,152.264
C04347=1097.646,274.282,-77.991,178.130,18.162,152.264
C04348=1097.652,274.530,-78.019,178.133,18.163,152.264
C04349=1097.658,274.778,-78.048,178.136,18.165,152.264
C04350=1097.663,275.027,-78.077,178.140,18.167,152.263
C04351=1097.669,275.275,-78.106,178.143,18.168,152.263
C04352=1097.675,275.524,-78.134,178.147,18.170,152.263
C04353=1097.683,275.884,-78.176,178.151,18.172,152.263
C04354=1097.691,276.245,-78.218,178.156,18.175,152.262
C04355=1097.699,276.606,-78.260,178.161,18.177,152.262
C04356=1097.707,276.968,-78.302,178.166,18.180,152.262
C04357=1097.713,277.216,-78.330,178.169,18.182,152.261
C04358=1097.719,277.464,-78.359,178.172,18.184,152.261
C04359=1097.724,277.712,-78.389,178.176,18.186,152.261
C04360=1097.730,277.960,-78.417,178.179,18.187,152.261
C04361=1097.736,278.209,-78.446,178.183,18.189,152.260
C04362=1097.741,278.458,-78.475,178.185,18.191,152.260
C04363=1097.747,278.705,-78.503,178.189,18.192,152.260
C04364=1097.752,278.954,-78.533,178.192,18.194,152.260
C04365=1097.758,279.202,-78.561,178.196,18.196,152.260
C04366=1097.763,279.450,-78.590,178.199,18.198,152.259
C04367=1097.769,279.698,-78.620,178.202,18.199,152.259
C04368=1097.776,279.946,-78.649,178.205,18.202,152.259
C04369=1097.781,280.195,-78.677,178.209,18.204,152.259
C04370=1097.787,280.443,-78.706,178.212,18.205,152.259
C04371=1097.792,280.691,-78.736,178.216,18.207,152.258
C04372=1097.798,280.939,-78.765,178.219,18.209,152.258
C04373=1097.803,281.188,-78.793,178.222,18.210,152.258
C04374=1097.809,281.436,-78.822,178.226,18.212,152.258
C04375=1097.815,281.684,-78.852,178.229,18.214,152.257
C04376=1097.821,281.932,-78.881,178.233,18.216,152.257
C04377=1097.826,282.180,-78.910,178.235,18.218,152.257
C04378=1097.831,282.429,-78.940,178.238,18.220,152.257
C04379=1097.837,282.677,-78.968,178.242,18.222,152.257
C04380=1097.843,282.926,-78.998,178.245,18.223,152.256
C04381=1097.848,283.173,-79.027,178.249,18.225,152.256
C04382=1097.854,283.422,-79.056,178.252,18.227,152.256
C04383=1097.860,283.670,-79.086,178.255,18.229,152.256
C04384=1097.866,283.918,-79.115,178.258,18.231,152.256
C04385=1097.871,284.166,-79.144,178.262,18.233,152.256
C04386=1097.876,284.414,-79.174,178.265,18.235,152.255
C04387=1097.882,284.663,-79.203,178.269,18.236,152.255
C04388=1097.888,284.911,-79.233,178.272,18.239,152.255
C04389=1097.893,285.159,-79.262,178.275,18.240,152.255
C04390=1097.899,285.407,-79.291,178.278,18.242,152.255
C04391=1097.905,285.655,-79.320,178.282,18.244,152.254
C04392=1097.910,285.904,-79.350,178.285,18.246,152.254
C04393=1097.916,286.152,-79.379,178.289,18.248,152.254
C04394=1097.922,286.400,-79.409,178.292,18.250,152.254
C04395=1097.927,286.648,-79.438,178.296,18.252,152.254
C04396=1097.933,286.896,-79.468,178.298,18.254,152.254
C04397=1097.939,287.144,-79.497,178.301,18.255,152.253
C04398=1097.944,287.392,-79.527,178.305,18.257,152.253
C04399=1097.950,287.641,-79.557,178.308,18.259,152.253
C04400=1097.956,287.889,-79.586,178.312,18.261,152.253
C04401=1097.962,288.138,-79.615,178.315,18.263,152.253
C04402=1097.967,288.385,-79.645,178.319,18.265,152.252
C04403=1097.972,288.633,-79.675,178.321,18.267,152.252
C04404=1097.979,288.881,-79.704,178.325,18.269,152.252
C04405=1097.987,289.252,-79.748,178.330,18.272,152.252
C04406=1097.996,289.622,-79.793,178.335,18.275,152.251
C04407=1098.004,289.992,-79.837,178.340,18.278,152.251
C04408=1098.012,290.364,-79.881,178.345,18.280,152.251
C04409=1098.018,290.611,-79.911,178.348,18.282,152.251
C04410=1098.024,290.859,-79.941,178.351,18.284,152.251
C04411=1098.030,291.107,-79.971,178.354,18.287,152.251
C04412=1098.035,291.356,-80.001,178.358,18.288,152.250
C04413=1098.041,291.604,-80.030,178.361,18.290,152.250
C04414=1098.047,291.852,-80.061,178.365,18.293,152.250
C04415=1098.052,292.100,-80.090,178.368,18.295,152.250
C04416=1098.058,292.348,-80.121,178.371,18.296,152.250
C04417=1098.063,292.597,-80.150,178.374,18.298,152.250
C04418=1098.068,292.844,-80.180,178.378,18.300,152.249
C04419=1098.074,293.092,-80.210,178.381,18.302,152.249
C04420=1098.080,293.341,-80.240,178.384,18.304,152.249
C04421=1098.085,293.589,-80.270,178.388,18.307,152.249
C04422=1098.091,293.837,-80.300,178.391,18.308,152.249
C04423=1098.097,294.085,-80.330,178.394,18.311,152.249
C04424=1098.102,294.333,-80.360,178.398,18.313,152.248
C04425=1098.108,294.581,-80.390,178.401,18.315,152.248
C04426=1098.114,294.829,-80.420,178.405,18.317,152.248
C04427=1098.119,295.077,-80.450,178.407,18.318,152.248
C04428=1098.125,295.325,-80.480,178.410,18.321,152.248
C04429=1098.131,295.574,-80.510,178.414,18.322,152.248
C04430=1098.137,295.821,-80.540,178.417,18.325,152.248
C04431=1098.142,296.069,-80.571,178.421,18.327,152.247
C04432=1098.148,296.318,-80.600,178.424,18.329,152.247
C04433=1098.154,296.565,-80.631,178.427,18.331,152.247
C04434=1098.160,296.813,-80.661,178.431,18.333,152.247
C04435=1098.165,297.062,-80.691,178.434,18.335,152.247
C04436=1098.171,297.310,-80.721,178.437,18.337,152.247
C04437=1098.177,297.558,-80.752,178.441,18.340,152.247
C04438=1098.182,297.806,-80.783,178.444,18.342,152.246
C04439=1098.188,298.055,-80.812,178.447,18.344,152.246
C04440=1098.194,298.302,-80.843,178.451,18.346,152.246
C04441=1098.200,298.550,-80.873,178.454,18.348,152.246
C04442=1098.205,298.798,-80.903,178.457,18.350,152.246
C04443=1098.210,299.047,-80.934,178.461,18.353,152.246
C04444=1098.216,299.295,-80.964,178.463,18.354,152.246
C04445=1098.222,299.543,-80.994,178.467,18.356,152.246
C04446=1098.227,299.791,-81.025,178.470,18.359,152.246
C04447=1098.233,300.038,-81.056,178.473,18.361,152.246
C04448=1098.238,300.286,-81.086,178.476,18.363,152.245
C04449=1098.244,300.534,-81.117,178.480,18.365,152.245
C04450=1098.249,300.782,-81.147,178.483,18.368,152.245
C04451=1098.255,301.031,-81.177,178.486,18.370,152.245
C04452=1098.260,301.279,-81.208,178.489,18.372,152.245
C04453=1098.266,301.527,-81.238,178.493,18.374,152.245
C04454=1098.272,301.774,-81.269,178.496,18.376,152.245
C04455=1098.277,302.023,-81.299,178.499,18.379,152.245
C04456=1098.282,302.270,-81.330,178.503,18.381,152.245
C04457=1098.291,302.654,-81.378,178.508,18.384,152.244
C04458=1098.300,303.040,-81.425,178.513,18.388,152.244
C04459=1098.309,303.424,-81.473,178.518,18.392,152.244
C04460=1098.317,303.808,-81.520,178.523,18.395,152.244
C04461=1098.323,304.056,-81.550,178.527,18.397,152.244
C04462=1098.328,304.304,-81.581,178.530,18.399,152.244
C04463=1098.335,304.552,-81.613,178.533,18.402,152.244
C04464=1098.340,304.800,-81.644,178.536,18.404,152.244
C04465=1098.346,305.048,-81.674,178.540,18.406,152.244
C04466=1098.351,305.296,-81.705,178.543,18.409,152.244
C04467=1098.357,305.544,-81.735,178.546,18.411,152.244
C04468=1098.362,305.792,-81.766,178.550,18.413,152.243
C04469=1098.368,306.040,-81.798,178.553,18.415,152.243
C04470=1098.374,306.288,-81.829,178.556,18.417,152.243
C04471=1098.379,306.536,-81.859,178.559,18.420,152.243
C04472=1098.384,306.784,-81.890,178.562,18.422,152.243
C04473=1098.391,307.032,-81.921,178.566,18.424,152.243
C04474=1098.396,307.280,-81.952,178.569,18.427,152.243
C04475=1098.402,307.528,-81.983,178.572,18.429,152.243
C04476=1098.407,307.775,-82.014,178.575,18.431,152.243
C04477=1098.414,308.024,-82.045,178.579,18.434,152.243
C04478=1098.419,308.272,-82.076,178.582,18.436,152.243
C04479=1098.425,308.519,-82.107,178.586,18.439,152.243
C04480=1098.430,308.767,-82.138,178.589,18.441,152.242
C04481=1098.437,309.016,-82.169,178.593,18.443,152.242
C04482=1098.442,309.263,-82.200,178.596,18.446,152.242
C04483=1098.448,309.511,-82.231,178.599,18.448,152.242
C04484=1098.454,309.759,-82.263,178.602,18.450,152.242
C04485=1098.459,310.007,-82.294,178.606,18.452,152.242
C04486=1098.465,310.255,-82.325,178.609,18.455,152.242
C04487=1098.471,310.504,-82.356,178.612,18.457,152.242
C04488=1098.477,310.751,-82.387,178.615,18.459,152.242
C04489=1098.482,310.999,-82.418,178.619,18.462,152.242
C04490=1098.488,311.247,-82.450,178.622,18.464,152.242
C04491=1098.494,311.495,-82.481,178.625,18.466,152.242
C04492=1098.500,311.743,-82.513,178.628,18.469,152.242
C04493=1098.505,311.991,-82.543,178.631,18.471,152.242
C04494=1098.511,312.238,-82.575,178.635,18.473,152.242
C04495=1098.517,312.487,-82.606,178.638,18.476,152.242
C04496=1098.523,312.734,-82.637,178.641,18.478,152.242
C04497=1098.529,312.983,-82.669,178.644,18.480,152.241
C04498=1098.534,313.231,-82.700,178.648,18.483,152.241
C04499=1098.540,313.478,-82.731,178.651,18.486,152.241
C04500=1098.546,313.727,-82.762,178.655,18.488,152.241
C04501=1098.551,313.974,-82.794,178.658,18.491,152.241
C04502=1098.558,314.222,-82.825,178.661,18.493,152.241
C04503=1098.563,314.470,-82.857,178.664,18.495,152.241
C04504=1098.569,314.719,-82.888,178.668,18.498,152.241
C04505=1098.574,314.966,-82.920,178.671,18.500,152.241
C04506=1098.581,315.214,-82.952,178.674,18.502,152.241
C04507=1098.586,315.462,-82.982,178.677,18.505,152.241
C04508=1098.592,315.710,-83.014,178.680,18.507,152.241
C04509=1098.600,316.097,-83.063,178.686,18.512,152.241
C04510=1098.609,316.483,-83.113,178.691,18.515,152.241
C04511=1098.617,316.871,-83.163,178.695,18.519,152.241
C04512=1098.626,317.258,-83.212,178.701,18.524,152.241
C04513=1098.632,317.506,-83.244,178.704,18.526,152.241
C04514=1098.637,317.753,-83.276,178.707,18.529,152.241
C04515=1098.643,318.001,-83.308,178.710,18.531,152.241
C04516=1098.649,318.249,-83.340,178.713,18.534,152.241
C04517=1098.655,318.497,-83.372,178.716,18.536,152.241
C04518=1098.660,318.745,-83.402,178.720,18.539,152.241
C04519=1098.666,318.994,-83.435,178.723,18.542,152.241
C04520=1098.671,319.241,-83.466,178.727,18.544,152.241
C04521=1098.677,319.489,-83.498,178.729,18.547,152.241
C04522=1098.682,319.737,-83.530,178.732,18.550,152.241
C04523=1098.688,319.985,-83.562,178.736,18.552,152.241
C04524=1098.693,320.233,-83.594,178.739,18.555,152.241
C04525=1098.699,320.481,-83.626,178.743,18.558,152.241
C04526=1098.704,320.729,-83.658,178.746,18.561,152.241
C04527=1098.710,320.977,-83.690,178.749,18.563,152.241
C04528=1098.716,321.224,-83.722,178.752,18.566,152.242
C04529=1098.722,321.472,-83.754,178.755,18.568,152.241
C04530=1098.727,321.719,-83.786,178.758,18.571,152.242
C04531=1098.733,321.968,-83.819,178.761,18.573,152.242
C04532=1098.738,322.215,-83.850,178.765,18.576,152.242
C04533=1098.744,322.464,-83.882,178.768,18.579,152.242
C04534=1098.750,322.712,-83.914,178.771,18.581,152.242
C04535=1098.755,322.959,-83.946,178.774,18.584,152.242
C04536=1098.762,323.207,-83.979,178.777,18.587,152.242
C04537=1098.766,323.455,-84.011,178.781,18.589,152.242
C04538=1098.772,323.703,-84.043,178.784,18.593,152.242
C04539=1098.778,323.951,-84.075,178.787,18.595,152.242
C04540=1098.784,324.198,-84.107,178.791,18.598,152.242
C04541=1098.790,324.446,-84.139,178.794,18.600,152.242
C04542=1098.795,324.695,-84.172,178.797,18.603,152.242
C04543=1098.801,324.942,-84.204,178.800,18.606,152.242
C04544=1098.807,325.190,-84.236,178.804,18.609,152.242
C04545=1098.813,325.438,-84.268,178.807,18.612,152.242
C04546=1098.818,325.686,-84.301,178.810,18.614,152.242
C04547=1098.824,325.934,-84.333,178.813,18.617,152.242
C04548=1098.830,326.182,-84.365,178.816,18.619,152.242
C04549=1098.836,326.429,-84.398,178.820,18.623,152.242
C04550=1098.841,326.677,-84.430,178.823,18.626,152.243
C04551=1098.847,326.925,-84.462,178.826,18.628,152.243
C04552=1098.853,327.173,-84.495,178.829,18.631,152.243
C04553=1098.858,327.421,-84.527,178.832,18.633,152.243
C04554=1098.864,327.668,-84.560,178.836,18.637,152.243
C04555=1098.870,327.917,-84.592,178.839,18.639,152.243
C04556=1098.876,328.164,-84.625,178.842,18.642,152.243
C04557=1098.881,328.412,-84.657,178.845,18.645,152.243
C04558=1098.887,328.660,-84.690,178.849,18.648,152.243
C04559=1098.893,328.908,-84.722,178.852,18.651,152.243
C04560=1098.899,329.156,-84.755,178.854,18.653,152.243
C04561=1098.908,329.536,-84.805,178.859,18.657,152.243
C04562=1098.917,329.916,-84.855,178.865,18.662,152.243
C04563=1098.925,330.295,-84.905,178.869,18.666,152.244
C04564=1098.934,330.675,-84.955,178.874,18.671,152.244
C04565=1098.940,330.923,-84.988,178.877,18.673,152.244
C04566=1098.946,331.170,-85.020,178.880,18.676,152.244
C04567=1098.952,331.418,-85.052,178.884,18.679,152.244
C04568=1098.957,331.666,-85.086,178.887,18.682,152.244
C04569=1098.963,331.914,-85.118,178.890,18.685,152.244
C04570=1098.969,332.162,-85.151,178.893,18.688,152.244
C04571=1098.975,332.410,-85.184,178.897,18.691,152.244
C04572=1098.981,332.658,-85.217,178.900,18.694,152.244
C04573=1098.986,332.905,-85.250,178.903,18.697,152.245
C04574=1098.991,333.153,-85.282,178.907,18.700,152.245
C04575=1098.997,333.401,-85.315,178.909,18.703,152.245
C04576=1099.003,333.649,-85.348,178.912,18.706,152.245
C04577=1099.009,333.897,-85.382,178.916,18.709,152.245
C04578=1099.015,334.144,-85.414,178.919,18.712,152.245
C04579=1099.020,334.392,-85.447,178.922,18.715,152.245
C04580=1099.025,334.640,-85.480,178.925,18.718,152.246
C04581=1099.032,334.888,-85.513,178.929,18.721,152.246
C04582=1099.037,335.136,-85.546,178.932,18.724,152.246
C04583=1099.043,335.383,-85.579,178.934,18.727,152.246
C04584=1099.049,335.631,-85.612,178.938,18.730,152.246
C04585=1099.055,335.879,-85.645,178.941,18.733,152.246
C04586=1099.060,336.126,-85.678,178.944,18.736,152.246
C04587=1099.065,336.374,-85.712,178.948,18.740,152.247
C04588=1099.071,336.622,-85.744,178.951,18.742,152.247
C04589=1099.077,336.870,-85.778,178.953,18.746,152.247
C04590=1099.083,337.117,-85.811,178.957,18.749,152.247
C04591=1099.089,337.365,-85.844,178.960,18.752,152.247
C04592=1099.094,337.613,-85.877,178.963,18.755,152.247
C04593=1099.100,337.861,-85.911,178.967,18.758,152.247
C04594=1099.105,338.109,-85.944,178.969,18.761,152.248
C04595=1099.112,338.356,-85.977,178.972,18.764,152.248
C04596=1099.117,338.604,-86.010,178.976,18.768,152.248
C04597=1099.123,338.852,-86.044,178.979,18.771,152.248
C04598=1099.129,339.099,-86.077,178.982,18.774,152.248
C04599=1099.134,339.347,-86.111,178.985,18.777,152.249
C04600=1099.140,339.595,-86.144,178.988,18.780,152.249
C04601=1099.146,339.842,-86.176,178.991,18.784,152.249
C04602=1099.151,340.090,-86.210,178.995,18.787,152.249
C04603=1099.157,340.337,-86.244,178.997,18.790,152.249
C04604=1099.163,340.585,-86.277,179.001,18.794,152.250
C04605=1099.168,340.833,-86.310,179.004,18.797,152.250
C04606=1099.174,341.081,-86.344,179.007,18.800,152.250
C04607=1099.180,341.328,-86.378,179.010,18.804,152.250
C04608=1099.185,341.576,-86.411,179.013,18.806,152.250
C04609=1099.191,341.824,-86.445,179.017,18.810,152.251
C04610=1099.196,342.071,-86.479,179.019,18.813,152.251
C04611=1099.202,342.319,-86.512,179.022,18.816,152.251
C04612=1099.208,342.567,-86.545,179.026,18.820,152.251
C04613=1099.217,342.941,-86.596,179.030,18.824,152.252
C04614=1099.226,343.315,-86.647,179.035,18.830,152.252
C04615=1099.234,343.688,-86.698,179.040,18.835,152.252
C04616=1099.243,344.063,-86.749,179.044,18.839,152.253
C04617=1099.249,344.310,-86.783,179.048,18.843,152.253
C04618=1099.254,344.558,-86.816,179.051,18.846,152.253
C04619=1099.260,344.805,-86.850,179.054,18.850,152.253
C04620=1099.266,345.053,-86.883,179.057,18.853,152.253
C04621=1099.272,345.300,-86.917,179.061,18.857,152.254
C04622=1099.277,345.548,-86.951,179.063,18.860,152.254
C04623=1099.283,345.795,-86.985,179.066,18.863,152.254
C04624=1099.289,346.044,-87.019,179.070,18.867,152.254
C04625=1099.294,346.292,-87.053,179.072,18.870,152.255
C04626=1099.300,346.540,-87.086,179.076,18.874,152.255
C04627=1099.306,346.787,-87.121,179.078,18.877,152.255
C04628=1099.312,347.034,-87.155,179.082,18.881,152.256
C04629=1099.317,347.282,-87.188,179.085,18.884,152.256
C04630=1099.323,347.529,-87.222,179.088,18.888,152.256
C04631=1099.328,347.777,-87.257,179.091,18.891,152.256
C04632=1099.334,348.025,-87.290,179.095,18.895,152.257
C04633=1099.340,348.273,-87.324,179.097,18.898,152.257
C04634=1099.346,348.520,-87.358,179.101,18.902,152.257
C04635=1099.351,348.768,-87.393,179.103,18.905,152.257
C04636=1099.357,349.016,-87.426,179.107,18.909,152.258
C04637=1099.362,349.263,-87.460,179.110,18.912,152.258
C04638=1099.368,349.510,-87.495,179.113,18.917,152.258
C04639=1099.374,349.758,-87.530,179.116,18.920,152.259
C04640=1099.380,350.006,-87.564,179.119,18.923,152.259
C04641=1099.386,350.253,-87.598,179.122,18.927,152.259
C04642=1099.391,350.501,-87.631,179.125,18.931,152.260
C04643=1099.396,350.748,-87.666,179.128,18.934,152.260
C04644=1099.402,350.996,-87.700,179.131,18.938,152.260
C04645=1099.409,351.244,-87.734,179.134,18.941,152.260
C04646=1099.414,351.491,-87.769,179.138,18.945,152.261
C04647=1099.420,351.739,-87.803,179.140,18.949,152.261
C04648=1099.426,351.986,-87.837,179.144,18.952,152.261
C04649=1099.431,352.234,-87.872,179.146,18.956,152.262
C04650=1099.437,352.481,-87.906,179.150,18.960,152.262
C04651=1099.443,352.729,-87.940,179.152,18.963,152.262
C04652=1099.448,352.976,-87.975,179.156,18.967,152.263
C04653=1099.455,353.224,-88.009,179.158,18.971,152.263
C04654=1099.460,353.472,-88.044,179.162,18.974,152.263
C04655=1099.466,353.719,-88.078,179.164,18.978,152.264
C04656=1099.472,353.967,-88.112,179.168,18.982,152.264
C04657=1099.477,354.215,-88.147,179.171,18.986,152.264
C04658=1099.483,354.462,-88.181,179.174,18.990,152.265
C04659=1099.489,354.709,-88.216,179.177,18.993,152.265
C04660=1099.494,354.956,-88.250,179.180,18.997,152.265
C04661=1099.500,355.205,-88.285,179.183,19.001,152.266
C04662=1099.506,355.452,-88.319,179.186,19.005,152.266
C04663=1099.511,355.700,-88.354,179.189,19.008,152.267
C04664=1099.516,355.947,-88.389,179.192,19.013,152.267
C04665=1099.526,356.323,-88.442,179.197,19.019,152.268
C04666=1099.534,356.699,-88.494,179.202,19.024,152.268
C04667=1099.543,357.075,-88.547,179.206,19.030,152.269
C04668=1099.552,357.451,-88.599,179.211,19.036,152.269
C04669=1099.557,357.699,-88.634,179.213,19.040,152.270
C04670=1099.564,357.946,-88.669,179.217,19.044,152.270
C04671=1099.569,358.194,-88.704,179.219,19.047,152.270
C04672=1099.574,358.442,-88.739,179.223,19.051,152.271
C04673=1099.581,358.689,-88.774,179.226,19.056,152.271
C04674=1099.586,358.937,-88.809,179.228,19.059,152.272
C04675=1099.592,359.184,-88.844,179.232,19.063,152.272
C04676=1099.598,359.431,-88.878,179.234,19.067,152.272
C04677=1099.604,359.679,-88.914,179.237,19.071,152.273
C04678=1099.610,359.926,-88.948,179.241,19.076,152.273
C04679=1099.616,360.174,-88.984,179.243,19.079,152.274
C04680=1099.621,360.421,-89.018,179.246,19.083,152.274
C04681=1099.626,360.668,-89.054,179.250,19.088,152.275
C04682=1099.633,360.916,-89.088,179.252,19.091,152.275
C04683=1099.638,361.163,-89.123,179.255,19.096,152.276
C04684=1099.643,361.411,-89.158,179.259,19.100,152.276
C04685=1099.649,361.659,-89.194,179.261,19.104,152.276
C04686=1099.655,361.906,-89.228,179.264,19.108,152.277
C04687=1099.661,362.154,-89.264,179.267,19.112,152.277
C04688=1099.666,362.400,-89.299,179.270,19.116,152.278
C04689=1099.672,362.649,-89.334,179.273,19.120,152.278
C04690=1099.678,362.895,-89.369,179.276,19.125,152.279
C04691=1099.684,363.142,-89.404,179.279,19.128,152.279
C04692=1099.690,363.391,-89.439,179.282,19.133,152.280
C04693=1099.695,363.638,-89.474,179.285,19.137,152.280
C04694=1099.701,363.885,-89.510,179.288,19.141,152.281
C04695=1099.706,364.132,-89.546,179.291,19.145,152.281
C04696=1099.713,364.380,-89.580,179.294,19.150,152.282
C04697=1099.718,364.627,-89.615,179.296,19.153,152.282
C04698=1099.724,364.875,-89.651,179.300,19.158,152.283
C04699=1099.730,365.122,-89.686,179.303,19.162,152.283
C04700=1099.736,365.370,-89.722,179.306,19.167,152.284
C04701=1099.741,365.617,-89.757,179.308,19.171,152.284
C04702=1099.747,365.865,-89.793,179.311,19.175,152.284
C04703=1099.752,366.112,-89.828,179.315,19.179,152.285
C04704=1099.758,366.360,-89.864,179.318,19.184,152.286
C04705=1099.764,366.607,-89.899,179.320,19.188,152.286
C04706=1099.770,366.854,-89.935,179.323,19.192,152.287
C04707=1099.775,367.101,-89.970,179.326,19.197,152.287
C04708=1099.781,367.349,-90.006,179.329,19.201,152.288
C04709=1099.787,367.596,-90.041,179.332,19.205,152.288
C04710=1099.793,367.843,-90.077,179.335,19.210,152.289
C04711=1099.798,368.090,-90.112,179.338,19.214,152.289
C04712=1099.804,368.338,-90.148,179.341,19.219,152.290
C04713=1099.810,368.585,-90.183,179.343,19.223,152.290
C04714=1099.816,368.833,-90.219,179.346,19.227,152.291
C04715=1099.821,369.080,-90.254,179.349,19.232,152.292
C04716=1099.827,369.327,-90.290,179.352,19.237,152.292
C04717=1099.833,369.605,-90.331,179.355,19.242,152.293
C04718=1099.840,369.881,-90.370,179.358,19.246,152.293
C04719=1099.846,370.158,-90.411,179.362,19.252,152.294
C04720=1099.853,370.435,-90.451,179.365,19.256,152.295
C04721=1099.858,370.682,-90.487,179.368,19.261,152.295
C04722=1099.864,370.930,-90.523,179.371,19.266,152.296
C04723=1099.869,371.177,-90.558,179.373,19.270,152.296
C04724=1099.875,371.425,-90.594,179.376,19.274,152.297
C04725=1099.882,371.672,-90.630,179.379,19.279,152.298
C04726=1099.887,371.919,-90.665,179.382,19.284,152.298
C04727=1099.893,372.167,-90.702,179.385,19.289,152.299
C04728=1099.899,372.414,-90.738,179.388,19.293,152.299
C04729=1099.904,372.661,-90.774,179.391,19.298,152.300
C04730=1099.910,372.908,-90.809,179.394,19.302,152.301
C04731=1099.916,373.155,-90.845,179.396,19.307,152.301
C04732=1099.922,373.402,-90.881,179.400,19.312,152.302
C04733=1099.927,373.650,-90.917,179.403,19.316,152.302
C04734=1099.934,373.897,-90.954,179.405,19.321,152.303
C04735=1099.939,374.144,-90.989,179.408,19.325,152.304
C04736=1099.946,374.391,-91.026,179.411,19.330,152.304
C04737=1099.951,374.639,-91.062,179.413,19.335,152.305
C04738=1099.957,374.886,-91.098,179.417,19.340,152.306
C04739=1099.963,375.134,-91.134,179.419,19.345,152.306
C04740=1099.968,375.381,-91.171,179.422,19.350,152.307
C04741=1099.974,375.628,-91.206,179.425,19.355,152.308
C04742=1099.979,375.875,-91.243,179.427,19.359,152.308
C04743=1099.985,376.123,-91.279,179.430,19.364,152.309
C04744=1099.990,376.370,-91.316,179.433,19.369,152.310
C04745=1099.996,376.617,-91.351,179.436,19.374,152.310
C04746=1100.003,376.864,-91.388,179.439,19.379,152.311
C04747=1100.008,377.111,-91.425,179.442,19.384,152.312
C04748=1100.014,377.359,-91.460,179.445,19.389,152.313
C04749=1100.019,377.606,-91.497,179.447,19.393,152.313
C04750=1100.025,377.852,-91.533,179.450,19.398,152.314
C04751=1100.030,378.100,-91.570,179.453,19.403,152.315
C04752=1100.037,378.347,-91.606,179.456,19.408,152.315
C04753=1100.042,378.595,-91.643,179.459,19.413,152.316
C04754=1100.048,378.841,-91.679,179.461,19.418,152.317
C04755=1100.053,379.089,-91.716,179.464,19.423,152.317
C04756=1100.060,379.336,-91.752,179.466,19.428,152.318
C04757=1100.065,379.583,-91.789,179.469,19.433,152.319
C04758=1100.071,379.831,-91.826,179.472,19.438,152.320
C04759=1100.076,380.077,-91.862,179.475,19.443,152.320
C04760=1100.083,380.325,-91.898,179.478,19.448,152.321
C04761=1100.091,380.686,-91.952,179.482,19.455,152.322
C04762=1100.100,381.047,-92.005,179.486,19.463,152.323
C04763=1100.108,381.409,-92.059,179.490,19.471,152.324
C04764=1100.117,381.770,-92.113,179.494,19.478,152.326
C04765=1100.123,382.017,-92.149,179.497,19.483,152.326
C04766=1100.128,382.264,-92.186,179.499,19.489,152.327
C04767=1100.134,382.511,-92.222,179.502,19.493,152.328
C04768=1100.140,382.759,-92.259,179.505,19.499,152.329
C04769=1100.150,383.176,-92.322,179.510,19.508,152.330
C04770=1100.160,383.595,-92.385,179.514,19.517,152.331
C04771=1100.169,384.013,-92.447,179.519,19.526,152.333
C04772=1100.178,384.431,-92.509,179.523,19.535,152.334
C04773=1100.184,384.678,-92.546,179.526,19.540,152.335
C04774=1100.190,384.925,-92.584,179.528,19.545,152.336
C04775=1100.195,385.172,-92.621,179.531,19.551,152.337
C04776=1100.202,385.420,-92.657,179.534,19.556,152.338
C04777=1100.207,385.667,-92.694,179.537,19.562,152.338
C04778=1100.213,385.914,-92.731,179.540,19.568,152.339
C04779=1100.218,386.160,-92.769,179.542,19.573,152.340
C04780=1100.224,386.408,-92.806,179.545,19.578,152.341
C04781=1100.230,386.655,-92.843,179.547,19.584,152.342
C04782=1100.236,386.901,-92.880,179.550,19.589,152.343
C04783=1100.242,387.149,-92.917,179.553,19.595,152.344
C04784=1100.247,387.396,-92.954,179.555,19.600,152.345
C04785=1100.253,387.643,-92.992,179.558,19.606,152.345
C04786=1100.259,387.890,-93.029,179.560,19.611,152.346
C04787=1100.264,388.138,-93.066,179.564,19.617,152.347
C04788=1100.270,388.384,-93.104,179.566,19.623,152.348
C04789=1100.277,388.631,-93.140,179.569,19.629,152.349
C04790=1100.283,388.878,-93.178,179.572,19.634,152.350
C04791=1100.288,389.126,-93.215,179.574,19.640,152.351
C04792=1100.294,389.372,-93.253,179.577,19.645,152.352
C04793=1100.300,389.620,-93.290,179.579,19.651,152.353
C04794=1100.306,389.866,-93.327,179.582,19.657,152.354
C04795=1100.311,390.114,-93.364,179.585,19.663,152.355
C04796=1100.317,390.361,-93.402,179.588,19.668,152.355
C04797=1100.323,390.608,-93.439,179.590,19.674,152.356
C04798=1100.329,390.855,-93.477,179.592,19.680,152.357
C04799=1100.335,391.101,-93.515,179.595,19.685,152.358
C04800=1100.340,391.349,-93.552,179.597,19.691,152.359
C04801=1100.346,391.595,-93.589,179.601,19.697,152.360
C04802=1100.352,391.843,-93.626,179.603,19.703,152.361
C04803=1100.358,392.090,-93.665,179.606,19.709,152.362
C04804=1100.364,392.337,-93.702,179.608,19.714,152.363
C04805=1100.370,392.584,-93.739,179.610,19.720,152.364
C04806=1100.376,392.831,-93.777,179.614,19.726,152.365
C04807=1100.381,393.078,-93.815,179.616,19.732,152.366
C04808=1100.387,393.325,-93.853,179.619,19.738,152.367
C04809=1100.393,393.572,-93.890,179.621,19.744,152.368
C04810=1100.398,393.819,-93.928,179.623,19.750,152.369
C04811=1100.404,394.066,-93.966,179.626,19.756,152.370
C04812=1100.411,394.313,-94.004,179.629,19.762,152.371
C04813=1100.416,394.560,-94.042,179.631,19.768,152.372
C04814=1100.422,394.807,-94.079,179.633,19.774,152.373
C04815=1100.427,395.054,-94.117,179.637,19.780,152.374
C04816=1100.433,395.301,-94.155,179.639,19.786,152.375
C04817=1100.439,395.548,-94.193,179.641,19.792,152.377
C04818=1100.446,395.795,-94.231,179.644,19.798,152.378
C04819=1100.451,396.042,-94.269,179.647,19.805,152.379
C04820=1100.457,396.289,-94.307,179.649,19.811,152.380
C04821=1100.461,396.504,-94.340,179.652,19.816,152.381
C04822=1100.467,396.720,-94.373,179.653,19.822,152.382
C04823=1100.471,396.935,-94.406,179.656,19.827,152.383
C04824=1100.477,397.151,-94.439,179.657,19.833,152.384
C04825=1100.481,397.366,-94.472,179.660,19.838,152.385
C04826=1100.486,397.581,-94.506,179.663,19.844,152.386
C04827=1100.492,397.796,-94.539,179.664,19.849,152.387
C04828=1100.496,398.012,-94.572,179.667,19.855,152.388
C04829=1100.503,398.259,-94.610,179.669,19.861,152.389
C04830=1100.508,398.506,-94.648,179.671,19.867,152.390
C04831=1100.514,398.753,-94.686,179.674,19.874,152.391
C04832=1100.520,399.000,-94.724,179.676,19.880,152.392
C04833=1100.526,399.247,-94.763,179.679,19.887,152.393
C04834=1100.532,399.493,-94.801,179.682,19.893,152.394
C04835=1100.537,399.741,-94.839,179.684,19.899,152.396
C04836=1100.544,399.988,-94.877,179.687,19.906,152.397
C04837=1100.549,400.235,-94.916,179.689,19.912,152.398
C04838=1100.555,400.481,-94.954,179.691,19.919,152.399
C04839=1100.560,400.728,-94.993,179.694,19.926,152.400
C04840=1100.567,400.976,-95.031,179.696,19.932,152.401
C04841=1100.572,401.223,-95.069,179.699,19.939,152.403
C04842=1100.578,401.469,-95.108,179.701,19.945,152.404
C04843=1100.584,401.717,-95.146,179.703,19.952,152.405
C04844=1100.590,401.963,-95.184,179.706,19.959,152.406
C04845=1100.595,402.210,-95.223,179.708,19.965,152.408
C04846=1100.601,402.458,-95.262,179.711,19.972,152.409
C04847=1100.607,402.704,-95.300,179.713,19.979,152.410
C04848=1100.613,402.951,-95.339,179.716,19.986,152.411
C04849=1100.619,403.198,-95.377,179.718,19.992,152.413
C04850=1100.624,403.445,-95.416,179.720,19.999,152.414
C04851=1100.630,403.692,-95.455,179.723,20.006,152.415
C04852=1100.636,403.938,-95.493,179.725,20.012,152.416
C04853=1100.642,404.186,-95.532,179.728,20.020,152.418
C04854=1100.648,404.432,-95.570,179.730,20.026,152.419
C04855=1100.653,404.679,-95.609,179.733,20.033,152.420
C04856=1100.659,404.927,-95.648,179.735,20.040,152.422
C04857=1100.665,405.174,-95.686,179.738,20.047,152.423
C04858=1100.671,405.420,-95.725,179.740,20.054,152.424
C04859=1100.677,405.667,-95.763,179.742,20.061,152.425
C04860=1100.683,405.915,-95.803,179.745,20.068,152.427
C04861=1100.688,406.161,-95.842,179.747,20.075,152.428
C04862=1100.695,406.408,-95.880,179.750,20.082,152.429
C04863=1100.700,406.655,-95.919,179.752,20.089,152.431
C04864=1100.706,406.901,-95.958,179.754,20.097,152.432
C04865=1100.711,407.149,-95.997,179.756,20.104,152.434
C04866=1100.717,407.396,-96.036,179.759,20.111,152.435
C04867=1100.724,407.642,-96.075,179.762,20.118,152.436
C04868=1100.729,407.889,-96.114,179.763,20.125,152.438
C04869=1100.735,408.137,-96.153,179.766,20.132,152.439
C04870=1100.740,408.383,-96.192,179.768,20.139,152.440
C04871=1100.746,408.630,-96.231,179.771,20.147,152.442
C04872=1100.752,408.877,-96.270,179.773,20.154,152.443
C04873=1100.758,409.124,-96.310,179.775,20.161,152.445
C04874=1100.763,409.370,-96.349,179.778,20.169,152.446
C04875=1100.769,409.618,-96.387,179.780,20.177,152.448
C04876=1100.775,409.864,-96.426,179.782,20.184,152.449
C04877=1100.780,410.079,-96.460,179.784,20.190,152.450
C04878=1100.785,410.295,-96.495,179.786,20.197,152.452
C04879=1100.790,410.511,-96.530,179.788,20.204,152.453
C04880=1100.796,410.726,-96.564,179.790,20.210,152.454
C04881=1100.801,410.941,-96.598,179.792,20.217,152.455
C04882=1100.806,411.157,-96.633,179.794,20.223,152.457
C04883=1100.811,411.371,-96.666,179.796,20.230,152.458
C04884=1100.815,411.587,-96.701,179.798,20.236,152.459
C04885=1100.822,411.834,-96.740,179.801,20.244,152.461
C04886=1100.828,412.081,-96.780,179.804,20.252,152.462
C04887=1100.833,412.327,-96.819,179.805,20.259,152.464
C04888=1100.839,412.575,-96.858,179.808,20.267,152.465
C04889=1100.845,412.821,-96.897,179.810,20.275,152.467
C04890=1100.851,413.068,-96.937,179.813,20.283,152.468
C04891=1100.857,413.315,-96.977,179.815,20.290,152.470
C04892=1100.862,413.561,-97.017,179.817,20.298,152.471
C04893=1100.868,413.809,-97.056,179.819,20.306,152.473
C04894=1100.874,414.056,-97.095,179.822,20.314,152.475
C04895=1100.880,414.302,-97.135,179.824,20.322,152.476
C04896=1100.886,414.549,-97.175,179.827,20.330,152.478
C04897=1100.892,414.796,-97.214,179.828,20.337,152.479
C04898=1100.897,415.042,-97.253,179.831,20.345,152.481
C04899=1100.904,415.289,-97.293,179.833,20.353,152.483
C04900=1100.910,415.536,-97.333,179.835,20.361,152.484
C04901=1100.915,415.783,-97.373,179.838,20.369,152.486
C04902=1100.921,416.029,-97.413,179.840,20.377,152.487
C04903=1100.927,416.276,-97.452,179.843,20.385,152.489
C04904=1100.933,416.523,-97.492,179.845,20.394,152.491
C04905=1100.939,416.769,-97.531,179.846,20.401,152.492
C04906=1100.944,417.016,-97.572,179.849,20.409,152.494
C04907=1100.951,417.263,-97.611,179.851,20.418,152.496
C04908=1100.957,417.510,-97.651,179.853,20.426,152.497
C04909=1100.962,417.756,-97.691,179.855,20.434,152.499
C04910=1100.968,418.003,-97.731,179.858,20.443,152.501
C04911=1100.973,418.250,-97.771,179.860,20.451,152.502
C04912=1100.979,418.496,-97.811,179.862,20.459,152.504
C04913=1100.986,418.743,-97.851,179.864,20.468,152.506
C04914=1100.991,418.990,-97.891,179.867,20.476,152.508
C04915=1100.997,419.237,-97.931,179.869,20.485,152.509
C04916=1101.004,419.483,-97.972,179.871,20.493,152.511
C04917=1101.008,419.730,-98.011,179.873,20.502,152.513
C04918=1101.015,419.976,-98.051,179.875,20.510,152.514
C04919=1101.020,420.223,-98.092,179.877,20.519,152.516
C04920=1101.026,420.470,-98.132,179.880,20.527,152.518
C04921=1101.032,420.717,-98.172,179.882,20.536,152.520
C04922=1101.038,420.963,-98.212,179.884,20.544,152.522
C04923=1101.044,421.210,-98.253,179.886,20.553,152.523
C04924=1101.050,421.456,-98.293,179.888,20.562,152.525
C04925=1101.056,421.703,-98.333,179.891,20.571,152.527
C04926=1101.062,421.950,-98.374,179.893,20.580,152.529
C04927=1101.068,422.197,-98.413,179.895,20.588,152.531
C04928=1101.073,422.443,-98.454,179.897,20.597,152.533
C04929=1101.079,422.690,-98.494,179.899,20.606,152.534
C04930=1101.085,422.936,-98.535,179.902,20.615,152.536
C04931=1101.091,423.183,-98.575,179.904,20.623,152.538
C04932=1101.097,423.430,-98.615,179.905,20.632,152.540
C04933=1101.103,423.652,-98.653,179.908,20.641,152.542
C04934=1101.107,423.874,-98.689,179.909,20.648,152.543
C04935=1101.113,424.096,-98.725,179.912,20.657,152.545
C04936=1101.118,424.318,-98.762,179.914,20.665,152.547
C04937=1101.123,424.540,-98.798,179.915,20.673,152.549
C04938=1101.129,424.763,-98.835,179.917,20.682,152.550
C04939=1101.134,424.985,-98.872,179.919,20.690,152.552
C04940=1101.139,425.207,-98.908,179.921,20.698,152.554
C04941=1101.145,425.453,-98.949,179.923,20.707,152.556
C04942=1101.150,425.700,-98.989,179.925,20.716,152.558
C04943=1101.157,425.946,-99.030,179.927,20.726,152.560
C04944=1101.163,426.193,-99.071,179.929,20.735,152.562
C04945=1101.168,426.440,-99.112,179.931,20.744,152.564
C04946=1101.174,426.687,-99.152,179.933,20.754,152.566
C04947=1101.181,426.933,-99.193,179.936,20.763,152.568
C04948=1101.186,427.179,-99.234,179.938,20.773,152.570
C04949=1101.192,427.426,-99.275,179.940,20.782,152.572
C04950=1101.198,427.672,-99.316,179.941,20.791,152.574
C04951=1101.203,427.919,-99.357,179.944,20.801,152.576
C04952=1101.210,428.165,-99.398,179.946,20.811,152.578
C04953=1101.216,428.412,-99.439,179.947,20.820,152.580
C04954=1101.221,428.659,-99.479,179.950,20.830,152.582
C04955=1101.227,428.905,-99.521,179.952,20.840,152.584
C04956=1101.233,429.152,-99.561,179.953,20.849,152.587
C04957=1101.240,429.398,-99.602,179.956,20.859,152.589
C04958=1101.245,429.645,-99.643,179.958,20.869,152.591
C04959=1101.251,429.891,-99.685,179.959,20.878,152.593
C04960=1101.257,430.137,-99.726,179.962,20.889,152.595
C04961=1101.263,430.384,-99.767,179.963,20.898,152.597
C04962=1101.269,430.630,-99.808,179.965,20.908,152.599
C04963=1101.274,430.877,-99.849,179.968,20.918,152.602
C04964=1101.280,431.123,-99.890,179.969,20.928,152.604
C04965=1101.286,431.369,-99.932,179.972,20.938,152.606
C04966=1101.292,431.615,-99.973,179.973,20.948,152.608
C04967=1101.298,431.862,-100.014,179.976,20.959,152.610
C04968=1101.304,432.108,-100.055,179.977,20.968,152.613
C04969=1101.310,432.355,-100.097,179.979,20.978,152.615
C04970=1101.316,432.602,-100.139,179.981,20.989,152.617
C04971=1101.322,432.848,-100.180,179.983,20.999,152.619
C04972=1101.328,433.095,-100.221,179.985,21.010,152.622
C04973=1101.334,433.341,-100.262,179.986,21.020,152.624
C04974=1101.340,433.587,-100.304,179.989,21.030,152.626
C04975=1101.345,433.833,-100.346,179.990,21.040,152.629
C04976=1101.351,434.080,-100.387,179.992,21.051,152.631
C04977=1101.357,434.326,-100.429,179.994,21.061,152.633
C04978=1101.363,434.572,-100.470,179.996,21.072,152.636
C04979=1101.369,434.819,-100.513,179.998,21.082,152.638
C04980=1101.375,435.065,-100.554,180.000,21.093,152.641
C04981=1101.381,435.312,-100.596,-179.998,21.104,152.643
C04982=1101.387,435.558,-100.637,-179.997,21.115,152.645
C04983=1101.393,435.804,-100.679,-179.995,21.125,152.648
C04984=1101.398,436.051,-100.721,-179.993,21.136,152.650
C04985=1101.404,436.297,-100.762,-179.991,21.147,152.653
C04986=1101.410,436.544,-100.804,-179.990,21.157,152.655
C04987=1101.415,436.790,-100.846,-179.988,21.169,152.657
C04988=1101.422,437.036,-100.888,-179.986,21.180,152.660
C04989=1101.430,437.406,-100.951,-179.983,21.196,152.664
C04990=1101.440,437.776,-101.014,-179.980,21.213,152.667
C04991=1101.449,438.147,-101.077,-179.978,21.230,152.671
C04992=1101.458,438.517,-101.140,-179.975,21.246,152.675
C04993=1101.463,438.763,-101.182,-179.974,21.257,152.678
C04994=1101.469,439.010,-101.224,-179.972,21.268,152.680
C04995=1101.476,439.256,-101.266,-179.970,21.280,152.683
C04996=1101.482,439.502,-101.308,-179.969,21.290,152.685
C04997=1101.487,439.748,-101.350,-179.967,21.302,152.688
C04998=1101.494,439.995,-101.392,-179.965,21.314,152.690
C04999=1101.500,440.240,-101.434,-179.963,21.325,152.693
C05000=1101.505,440.487,-101.476,-179.962,21.336,152.696
C05001=1101.512,440.733,-101.519,-179.960,21.348,152.698
C05002=1101.517,440.980,-101.561,-179.958,21.360,152.701
C05003=1101.523,441.225,-101.603,-179.956,21.371,152.704
C05004=1101.529,441.472,-101.645,-179.955,21.383,152.706
C05005=1101.535,441.718,-101.688,-179.954,21.395,152.709
C05006=1101.541,441.964,-101.731,-179.952,21.407,152.712
C05007=1101.546,442.210,-101.773,-179.950,21.418,152.715
C05008=1101.553,442.457,-101.815,-179.948,21.430,152.717
C05009=1101.559,442.703,-101.858,-179.947,21.442,152.720
C05010=1101.565,442.948,-101.900,-179.946,21.454,152.723
C05011=1101.571,443.195,-101.943,-179.944,21.466,152.726
C05012=1101.576,443.441,-101.985,-179.942,21.478,152.729
C05013=1101.582,443.687,-102.027,-179.941,21.490,152.731
C05014=1101.588,443.934,-102.071,-179.940,21.502,152.734
C05015=1101.594,444.179,-102.113,-179.938,21.514,152.737
C05016=1101.601,444.426,-102.155,-179.937,21.526,152.740
C05017=1101.606,444.672,-102.198,-179.937,21.538,152.743
C05018=1101.612,444.919,-102.241,-179.936,21.550,152.746
C05019=1101.618,445.164,-102.283,-179.935,21.562,152.749
C05020=1101.624,445.410,-102.326,-179.935,21.574,152.752
C05021=1101.630,445.657,-102.369,-179.934,21.586,152.755
C05022=1101.636,445.903,-102.412,-179.934,21.598,152.758
C05023=1101.642,446.149,-102.454,-179.935,21.610,152.761
C05024=1101.648,446.395,-102.497,-179.934,21.622,152.764
C05025=1101.654,446.642,-102.540,-179.934,21.634,152.767
C05026=1101.660,446.887,-102.583,-179.935,21.645,152.770
C05027=1101.666,447.134,-102.626,-179.935,21.657,152.773
C05028=1101.671,447.380,-102.669,-179.935,21.669,152.776
C05029=1101.677,447.627,-102.712,-179.936,21.681,152.779
C05030=1101.683,447.872,-102.755,-179.937,21.693,152.782
C05031=1101.690,448.119,-102.797,-179.938,21.705,152.785
C05032=1101.695,448.365,-102.840,-179.939,21.716,152.789
C05033=1101.702,448.611,-102.884,-179.940,21.728,152.792
C05034=1101.707,448.856,-102.927,-179.941,21.740,152.795
C05035=1101.713,449.103,-102.970,-179.942,21.751,152.798
C05036=1101.719,449.350,-103.013,-179.944,21.763,152.801
C05037=1101.725,449.596,-103.056,-179.945,21.775,152.805
C05038=1101.730,449.841,-103.099,-179.946,21.787,152.808
C05039=1101.737,450.087,-103.143,-179.949,21.798,152.811
C05040=1101.744,450.334,-103.185,-179.950,21.810,152.814
C05041=1101.344,450.326,-103.326,179.981,22.033,152.882
C05042=1101.337,450.080,-103.284,179.983,22.022,152.878
C05043=1101.331,449.833,-103.241,179.984,22.010,152.875
C05044=1101.325,449.588,-103.197,179.986,21.998,152.872
C05045=1101.319,449.341,-103.154,179.988,21.987,152.869
C05046=1101.314,449.095,-103.111,179.989,21.975,152.866
C05047=1101.307,448.849,-103.067,179.990,21.963,152.862
C05048=1101.302,448.604,-103.025,179.991,21.951,152.859
C05049=1101.296,448.357,-102.982,179.992,21.939,152.856
C05050=1101.290,448.110,-102.938,179.993,21.927,152.853
C05051=1101.284,447.864,-102.896,179.994,21.916,152.850
C05052=1101.278,447.618,-102.853,179.995,21.903,152.846
C05053=1101.271,447.373,-102.810,179.995,21.891,152.843
C05054=1101.265,447.126,-102.767,179.996,21.880,152.840
C05055=1101.260,446.880,-102.724,179.996,21.868,152.837
C05056=1101.254,446.634,-102.681,179.997,21.856,152.834
C05057=1101.248,446.388,-102.638,179.997,21.844,152.831
C05058=1101.242,446.141,-102.595,179.996,21.831,152.828
C05059=1101.236,445.895,-102.552,179.997,21.820,152.825
C05060=1101.230,445.649,-102.509,179.996,21.807,152.822
C05061=1101.224,445.403,-102.467,179.996,21.796,152.819
C05062=1101.218,445.157,-102.424,179.995,21.784,152.816
C05063=1101.212,444.911,-102.381,179.994,21.772,152.813
C05064=1101.206,444.664,-102.338,179.994,21.759,152.810
C05065=1101.200,444.419,-102.295,179.993,21.748,152.807
C05066=1101.194,444.172,-102.252,179.991,21.735,152.804
C05067=1101.188,443.926,-102.210,179.990,21.723,152.801
C05068=1101.182,443.681,-102.167,179.989,21.711,152.798
C05069=1101.176,443.434,-102.124,179.988,21.699,152.796
C05070=1101.171,443.188,-102.081,179.986,21.687,152.793
C05071=1101.164,442.941,-102.040,179.984,21.675,152.790
C05072=1101.159,442.695,-101.997,179.982,21.663,152.787
C05073=1101.152,442.450,-101.955,179.981,21.650,152.784
C05074=1101.146,442.203,-101.912,179.979,21.638,152.782
C05075=1101.141,441.957,-101.870,179.978,21.627,152.779
C05076=1101.135,441.711,-101.827,179.976,21.615,152.776
C05077=1101.129,441.464,-101.784,179.974,21.603,152.773
C05078=1101.122,441.219,-101.742,179.972,21.591,152.771
C05079=1101.116,440.972,-101.700,179.970,21.580,152.768
C05080=1101.110,440.726,-101.657,179.969,21.568,152.765
C05081=1101.105,440.479,-101.615,179.967,21.556,152.763
C05082=1101.099,440.234,-101.573,179.965,21.545,152.760
C05083=1101.093,439.987,-101.531,179.963,21.533,152.757
C05084=1101.087,439.741,-101.489,179.962,21.522,152.755
C05085=1101.080,439.496,-101.446,179.960,21.510,152.752
C05086=1101.075,439.248,-101.404,179.958,21.499,152.750
C05087=1101.069,439.002,-101.363,179.957,21.488,152.747
C05088=1101.063,438.756,-101.320,179.955,21.476,152.744
C05089=1101.057,438.509,-101.278,179.953,21.465,152.742
C05090=1101.048,438.146,-101.216,179.950,21.448,152.738
C05091=1101.039,437.783,-101.154,179.948,21.432,152.734
C05092=1101.030,437.419,-101.092,179.945,21.416,152.731
C05093=1101.021,437.057,-101.030,179.942,21.400,152.727
C05094=1101.016,436.810,-100.988,179.940,21.388,152.724
C05095=1101.009,436.563,-100.946,179.939,21.378,152.722
C05096=1101.003,436.317,-100.905,179.937,21.367,152.720
C05097=1100.998,436.071,-100.863,179.935,21.356,152.717
C05098=1100.992,435.825,-100.820,179.933,21.345,152.715
C05099=1100.986,435.579,-100.779,179.931,21.334,152.712
C05100=1100.980,435.333,-100.737,179.930,21.323,152.710
C05101=1100.974,435.086,-100.696,179.927,21.312,152.707
C05102=1100.968,434.839,-100.654,179.926,21.302,152.705
C05103=1100.962,434.593,-100.612,179.924,21.291,152.703
C05104=1100.956,434.347,-100.571,179.922,21.281,152.700
C05105=1100.951,434.101,-100.529,179.920,21.270,152.698
C05106=1100.945,433.854,-100.487,179.918,21.260,152.696
C05107=1100.939,433.608,-100.446,179.916,21.249,152.693
C05108=1100.933,433.362,-100.404,179.915,21.239,152.691
C05109=1100.927,433.115,-100.362,179.912,21.228,152.688
C05110=1100.921,432.869,-100.321,179.911,21.218,152.686
C05111=1100.915,432.622,-100.279,179.908,21.208,152.684
C05112=1100.909,432.376,-100.238,179.907,21.197,152.682
C05113=1100.903,432.129,-100.197,179.904,21.187,152.679
C05114=1100.897,431.883,-100.156,179.903,21.177,152.677
C05115=1100.891,431.637,-100.114,179.900,21.166,152.675
C05116=1100.886,431.391,-100.073,179.899,21.157,152.673
C05117=1100.879,431.144,-100.031,179.896,21.146,152.670
C05118=1100.873,430.897,-99.990,179.894,21.136,152.668
C05119=1100.867,430.651,-99.949,179.893,21.126,152.666
C05120=1100.861,430.405,-99.907,179.890,21.116,152.664
C05121=1100.856,430.158,-99.867,179.889,21.106,152.662
C05122=1100.850,429.912,-99.825,179.886,21.096,152.659
C05123=1100.844,429.665,-99.784,179.884,21.086,152.657
C05124=1100.838,429.419,-99.743,179.883,21.076,152.655
C05125=1100.832,429.172,-99.702,179.880,21.066,152.653
C05126=1100.827,428.926,-99.661,179.878,21.057,152.651
C05127=1100.821,428.679,-99.619,179.876,21.047,152.649
C05128=1100.815,428.433,-99.579,179.874,21.037,152.647
C05129=1100.808,428.187,-99.538,179.872,21.028,152.645
C05130=1100.803,427.940,-99.497,179.870,21.018,152.643
C05131=1100.797,427.694,-99.456,179.868,21.008,152.640
C05132=1100.791,427.447,-99.415,179.866,20.999,152.638
C05133=1100.785,427.201,-99.373,179.864,20.990,152.636
C05134=1100.779,426.954,-99.333,179.862,20.980,152.634
C05135=1100.773,426.707,-99.292,179.859,20.970,152.632
C05136=1100.767,426.461,-99.251,179.857,20.961,152.630
C05137=1100.762,426.214,-99.210,179.856,20.952,152.628
C05138=1100.755,425.968,-99.170,179.854,20.942,152.626
C05139=1100.750,425.721,-99.129,179.851,20.933,152.624
C05140=1100.744,425.475,-99.088,179.849,20.924,152.622
C05141=1100.738,425.228,-99.047,179.847,20.914,152.620
C05142=1100.733,425.005,-99.011,179.845,20.906,152.619
C05143=1100.727,424.783,-98.974,179.843,20.898,152.617
C05144=1100.722,424.561,-98.937,179.841,20.889,152.615
C05145=1100.716,424.338,-98.901,179.840,20.881,152.613
C05146=1100.711,424.115,-98.864,179.837,20.873,152.611
C05147=1100.706,423.892,-98.827,179.835,20.864,152.610
C05148=1100.701,423.670,-98.790,179.833,20.857,152.608
C05149=1100.695,423.448,-98.754,179.831,20.848,152.606
C05150=1100.690,423.202,-98.714,179.829,20.839,152.604
C05151=1100.684,422.955,-98.673,179.827,20.830,152.602
C05152=1100.678,422.708,-98.633,179.825,20.821,152.601
C05153=1100.672,422.462,-98.592,179.823,20.812,152.599
C05154=1100.666,422.215,-98.552,179.821,20.804,152.597
C05155=1100.660,421.969,-98.512,179.818,20.794,152.595
C05156=1100.654,421.722,-98.471,179.816,20.786,152.593
C05157=1100.648,421.475,-98.431,179.814,20.777,152.591
C05158=1100.643,421.229,-98.390,179.812,20.768,152.590
C05159=1100.637,420.982,-98.351,179.809,20.759,152.588
C05160=1100.631,420.735,-98.310,179.807,20.751,152.586
C05161=1100.625,420.489,-98.270,179.805,20.742,152.584
C05162=1100.618,420.242,-98.230,179.803,20.733,152.582
C05163=1100.613,419.995,-98.189,179.801,20.725,152.581
C05164=1100.607,419.749,-98.150,179.798,20.716,152.579
C05165=1100.602,419.502,-98.109,179.796,20.708,152.577
C05166=1100.595,419.256,-98.069,179.794,20.699,152.575
C05167=1100.590,419.009,-98.028,179.792,20.691,152.573
C05168=1100.584,418.762,-97.989,179.790,20.682,152.572
C05169=1100.578,418.516,-97.949,179.787,20.673,152.570
C05170=1100.572,418.269,-97.908,179.785,20.665,152.568
C05171=1100.566,418.022,-97.869,179.783,20.657,152.567
C05172=1100.560,417.775,-97.828,179.780,20.649,152.565
C05173=1100.555,417.529,-97.789,179.778,20.640,152.563
C05174=1100.549,417.282,-97.749,179.776,20.632,152.561
C05175=1100.543,417.035,-97.709,179.774,20.623,152.560
C05176=1100.537,416.788,-97.669,179.771,20.615,152.558
C05177=1100.531,416.542,-97.629,179.769,20.607,152.556
C05178=1100.526,416.295,-97.589,179.767,20.599,152.555
C05179=1100.520,416.048,-97.550,179.765,20.591,152.553
C05180=1100.513,415.801,-97.509,179.762,20.583,152.552
C05181=1100.508,415.555,-97.470,179.760,20.575,152.550
C05182=1100.501,415.308,-97.430,179.758,20.566,152.548
C05183=1100.495,415.061,-97.391,179.755,20.558,152.547
C05184=1100.491,414.814,-97.351,179.753,20.551,152.545
C05185=1100.484,414.568,-97.311,179.751,20.542,152.543
C05186=1100.478,414.321,-97.272,179.748,20.534,152.542
C05187=1100.472,414.074,-97.232,179.746,20.527,152.540
C05188=1100.466,413.828,-97.192,179.744,20.519,152.539
C05189=1100.460,413.581,-97.153,179.742,20.511,152.537
C05190=1100.454,413.333,-97.113,179.739,20.503,152.535
C05191=1100.449,413.087,-97.074,179.736,20.495,152.534
C05192=1100.442,412.840,-97.034,179.735,20.487,152.532
C05193=1100.436,412.593,-96.995,179.732,20.480,152.531
C05194=1100.431,412.347,-96.955,179.730,20.472,152.529
C05195=1100.425,412.099,-96.916,179.727,20.464,152.528
C05196=1100.420,411.853,-96.877,179.725,20.457,152.526
C05197=1100.414,411.606,-96.837,179.723,20.449,152.525
C05198=1100.409,411.390,-96.803,179.721,20.442,152.524
C05199=1100.403,411.175,-96.769,179.719,20.435,152.522
C05200=1100.398,410.960,-96.734,179.717,20.429,152.521
C05201=1100.393,410.743,-96.699,179.715,20.422,152.520
C05202=1100.388,410.528,-96.665,179.713,20.416,152.518
C05203=1100.383,410.312,-96.631,179.711,20.409,152.517
C05204=1100.378,410.097,-96.597,179.709,20.402,152.516
C05205=1100.373,409.881,-96.562,179.706,20.396,152.514
C05206=1100.367,409.634,-96.523,179.704,20.388,152.513
C05207=1100.361,409.387,-96.484,179.701,20.381,152.512
C05208=1100.355,409.140,-96.444,179.699,20.373,152.510
C05209=1100.350,408.894,-96.405,179.697,20.366,152.509
C05210=1100.344,408.646,-96.367,179.695,20.359,152.507
C05211=1100.339,408.400,-96.327,179.692,20.351,152.506
C05212=1100.333,408.153,-96.288,179.689,20.344,152.504
C05213=1100.327,407.906,-96.249,179.688,20.337,152.503
C05214=1100.320,407.659,-96.210,179.685,20.329,152.502
C05215=1100.315,407.413,-96.171,179.682,20.322,152.500
C05216=1100.309,407.165,-96.132,179.680,20.315,152.499
C05217=1100.304,406.919,-96.093,179.678,20.307,152.497
C05218=1100.297,406.672,-96.054,179.676,20.300,152.496
C05219=1100.292,406.425,-96.015,179.673,20.293,152.495
C05220=1100.286,406.178,-95.977,179.670,20.286,152.493
C05221=1100.280,405.931,-95.938,179.668,20.279,152.492
C05222=1100.275,405.685,-95.899,179.665,20.272,152.491
C05223=1100.269,405.437,-95.860,179.664,20.265,152.489
C05224=1100.263,405.191,-95.821,179.661,20.257,152.488
C05225=1100.257,404.943,-95.783,179.659,20.251,152.487
C05226=1100.251,404.697,-95.744,179.656,20.243,152.485
C05227=1100.245,404.450,-95.704,179.654,20.237,152.484
C05228=1100.239,404.203,-95.666,179.651,20.230,152.483
C05229=1100.233,403.956,-95.627,179.649,20.223,152.481
C05230=1100.228,403.709,-95.589,179.646,20.216,152.480
C05231=1100.222,403.463,-95.550,179.644,20.209,152.479
C05232=1100.216,403.215,-95.511,179.641,20.202,152.477
C05233=1100.210,402.969,-95.473,179.639,20.196,152.476
C05234=1100.204,402.721,-95.434,179.636,20.189,152.475
C05235=1100.199,402.474,-95.396,179.634,20.182,152.474
C05236=1100.193,402.228,-95.357,179.631,20.175,152.473
C05237=1100.187,401.980,-95.319,179.629,20.168,152.471
C05238=1100.181,401.734,-95.280,179.627,20.162,152.470
C05239=1100.175,401.486,-95.241,179.624,20.155,152.469
C05240=1100.169,401.239,-95.204,179.622,20.148,152.468
C05241=1100.164,400.993,-95.165,179.619,20.141,152.466
C05242=1100.158,400.745,-95.126,179.617,20.135,152.465
C05243=1100.152,400.498,-95.088,179.615,20.129,152.464
C05244=1100.147,400.251,-95.050,179.612,20.121,152.463
C05245=1100.141,400.005,-95.011,179.609,20.115,152.462
C05246=1100.135,399.757,-94.973,179.607,20.108,152.460
C05247=1100.129,399.511,-94.935,179.604,20.102,152.459
C05248=1100.124,399.264,-94.897,179.602,20.096,152.458
C05249=1100.117,399.016,-94.858,179.599,20.089,152.457
C05250=1100.111,398.770,-94.820,179.597,20.083,152.456
C05251=1100.106,398.523,-94.782,179.595,20.076,152.454
C05252=1100.099,398.276,-94.743,179.592,20.070,152.453
C05253=1100.094,398.029,-94.705,179.589,20.063,152.452
C05254=1100.089,397.813,-94.672,179.587,20.058,152.451
C05255=1100.084,397.598,-94.639,179.585,20.053,152.450
C05256=1100.079,397.382,-94.606,179.583,20.047,152.449
C05257=1100.074,397.166,-94.572,179.580,20.041,152.448
C05258=1100.069,396.951,-94.540,179.578,20.036,152.447
C05259=1100.064,396.735,-94.506,179.576,20.030,152.446
C05260=1100.059,396.520,-94.473,179.574,20.025,152.445
C05261=1100.053,396.304,-94.440,179.572,20.019,152.444
C05262=1100.048,396.057,-94.402,179.570,20.013,152.443
C05263=1100.042,395.810,-94.364,179.566,20.006,152.442
C05264=1100.036,395.563,-94.326,179.564,20.001,152.441
C05265=1100.031,395.316,-94.288,179.562,19.994,152.440
C05266=1100.025,395.069,-94.250,179.560,19.988,152.439
C05267=1100.019,394.822,-94.212,179.556,19.982,152.438
C05268=1100.013,394.576,-94.174,179.554,19.976,152.437
C05269=1100.007,394.329,-94.137,179.551,19.970,152.436
C05270=1100.002,394.080,-94.099,179.549,19.964,152.435
C05271=1099.996,393.834,-94.061,179.546,19.957,152.434
C05272=1099.990,393.587,-94.023,179.543,19.952,152.433
C05273=1099.984,393.340,-93.985,179.541,19.945,152.432
C05274=1099.978,393.093,-93.948,179.539,19.940,152.431
C05275=1099.972,392.846,-93.910,179.535,19.933,152.430
C05276=1099.967,392.599,-93.872,179.533,19.927,152.428
C05277=1099.961,392.352,-93.834,179.531,19.921,152.427
C05278=1099.955,392.105,-93.796,179.528,19.916,152.426
C05279=1099.949,391.857,-93.759,179.526,19.910,152.425
C05280=1099.943,391.611,-93.721,179.522,19.904,152.425
C05281=1099.937,391.364,-93.684,179.520,19.898,152.424
C05282=1099.932,391.117,-93.647,179.518,19.892,152.423
C05283=1099.926,390.870,-93.609,179.515,19.886,152.422
C05284=1099.920,390.622,-93.572,179.513,19.881,152.421
C05285=1099.914,390.376,-93.534,179.510,19.875,152.420
C05286=1099.909,390.129,-93.496,179.507,19.869,152.419
C05287=1099.903,389.882,-93.459,179.504,19.863,152.418
C05288=1099.896,389.635,-93.422,179.502,19.857,152.417
C05289=1099.891,389.388,-93.385,179.499,19.852,152.416
C05290=1099.885,389.141,-93.347,179.497,19.846,152.415
C05291=1099.879,388.894,-93.310,179.494,19.840,152.414
C05292=1099.873,388.647,-93.273,179.491,19.835,152.413
C05293=1099.868,388.400,-93.236,179.488,19.829,152.412
C05294=1099.862,388.153,-93.198,179.485,19.823,152.411
C05295=1099.856,387.906,-93.161,179.483,19.818,152.410
C05296=1099.851,387.658,-93.124,179.480,19.812,152.409
C05297=1099.845,387.411,-93.086,179.478,19.806,152.408
C05298=1099.838,387.164,-93.050,179.475,19.801,152.408
C05299=1099.832,386.918,-93.012,179.473,19.795,152.407
C05300=1099.827,386.670,-92.975,179.470,19.790,152.406
C05301=1099.821,386.423,-92.938,179.466,19.784,152.405
C05302=1099.815,386.176,-92.900,179.464,19.778,152.404
C05303=1099.810,385.929,-92.863,179.461,19.773,152.403
C05304=1099.803,385.682,-92.826,179.459,19.768,152.402
C05305=1099.798,385.434,-92.789,179.456,19.762,152.401
C05306=1099.792,385.188,-92.752,179.453,19.757,152.401
C05307=1099.787,384.941,-92.715,179.451,19.751,152.400
C05308=1099.781,384.694,-92.678,179.448,19.746,152.399
C05309=1099.775,384.447,-92.641,179.445,19.740,152.398
C05310=1099.770,384.237,-92.609,179.443,19.736,152.397
C05311=1099.766,384.027,-92.578,179.440,19.731,152.397
C05312=1099.761,383.819,-92.547,179.438,19.727,152.396
C05313=1099.756,383.609,-92.516,179.436,19.722,152.395
C05314=1099.751,383.400,-92.484,179.433,19.717,152.394
C05315=1099.746,383.191,-92.454,179.431,19.713,152.394
C05316=1099.736,382.772,-92.391,179.427,19.704,152.392
C05317=1099.731,382.524,-92.354,179.424,19.699,152.392
C05318=1099.725,382.277,-92.317,179.422,19.693,152.391
C05319=1099.719,382.030,-92.281,179.419,19.689,152.390
C05320=1099.714,381.783,-92.244,179.416,19.683,152.389
C05321=1099.707,381.536,-92.208,179.414,19.678,152.388
C05322=1099.702,381.289,-92.171,179.411,19.673,152.388
C05323=1099.696,381.042,-92.134,179.408,19.667,152.387
C05324=1099.690,380.794,-92.097,179.405,19.663,152.386
C05325=1099.684,380.547,-92.060,179.402,19.657,152.385
C05326=1099.678,380.300,-92.024,179.399,19.652,152.385
C05327=1099.673,380.053,-91.987,179.397,19.647,152.384
C05328=1099.667,379.806,-91.950,179.394,19.642,152.383
C05329=1099.661,379.558,-91.914,179.391,19.637,152.382
C05330=1099.655,379.311,-91.878,179.388,19.632,152.381
C05331=1099.649,379.064,-91.841,179.385,19.627,152.381
C05332=1099.644,378.818,-91.805,179.383,19.622,152.380
C05333=1099.638,378.570,-91.768,179.380,19.616,152.379
C05334=1099.632,378.323,-91.732,179.377,19.611,152.379
C05335=1099.626,378.075,-91.695,179.374,19.606,152.378
C05336=1099.621,377.829,-91.659,179.371,19.601,152.377
C05337=1099.615,377.581,-91.622,179.369,19.596,152.376
C05338=1099.609,377.334,-91.586,179.366,19.591,152.376
C05339=1099.603,377.086,-91.549,179.363,19.586,152.375
C05340=1099.598,376.840,-91.513,179.361,19.582,152.374
C05341=1099.592,376.592,-91.477,179.358,19.577,152.374
C05342=1099.586,376.345,-91.440,179.355,19.572,152.373
C05343=1099.581,376.098,-91.405,179.352,19.567,152.372
C05344=1099.575,375.851,-91.368,179.349,19.562,152.371
C05345=1099.569,375.604,-91.331,179.346,19.557,152.371
C05346=1099.564,375.356,-91.295,179.343,19.552,152.370
C05347=1099.558,375.109,-91.259,179.340,19.547,152.369
C05348=1099.552,374.862,-91.223,179.338,19.542,152.369
C05349=1099.547,374.615,-91.186,179.335,19.537,152.368
C05350=1099.541,374.367,-91.151,179.333,19.533,152.367
C05351=1099.534,374.120,-91.114,179.329,19.528,152.367
C05352=1099.530,373.873,-91.078,179.327,19.523,152.366
C05353=1099.524,373.625,-91.043,179.324,19.518,152.365
C05354=1099.517,373.378,-91.006,179.321,19.514,152.365
C05355=1099.511,373.131,-90.970,179.318,19.509,152.364
C05356=1099.505,372.884,-90.934,179.315,19.504,152.364
C05357=1099.500,372.636,-90.898,179.312,19.500,152.363
C05358=1099.494,372.389,-90.862,179.309,19.495,152.362
C05359=1099.488,372.142,-90.826,179.306,19.490,152.362
C05360=1099.482,371.895,-90.790,179.303,19.486,152.361
C05361=1099.476,371.647,-90.755,179.300,19.481,152.360
C05362=1099.471,371.400,-90.719,179.298,19.477,152.360
C05363=1099.465,371.152,-90.682,179.295,19.472,152.359
C05364=1099.460,370.906,-90.647,179.292,19.467,152.359
C05365=1099.450,370.514,-90.590,179.287,19.460,152.358
C05366=1099.441,370.122,-90.534,179.283,19.453,152.357
C05367=1099.433,369.731,-90.477,179.278,19.445,152.356
C05368=1099.423,369.339,-90.420,179.273,19.438,152.355
C05369=1099.417,369.092,-90.384,179.271,19.434,152.354
C05370=1099.411,368.845,-90.349,179.268,19.429,152.354
C05371=1099.406,368.597,-90.313,179.265,19.425,152.353
C05372=1099.401,368.350,-90.277,179.262,19.420,152.353
C05373=1099.395,368.102,-90.242,179.260,19.416,152.352
C05374=1099.389,367.855,-90.206,179.257,19.412,152.351
C05375=1099.383,367.608,-90.171,179.253,19.407,152.351
C05376=1099.377,367.360,-90.135,179.250,19.402,152.350
C05377=1099.372,367.113,-90.099,179.248,19.398,152.350
C05378=1099.366,366.865,-90.064,179.245,19.393,152.349
C05379=1099.360,366.618,-90.028,179.242,19.389,152.349
C05380=1099.354,366.371,-89.993,179.239,19.384,152.348
C05381=1099.349,366.124,-89.957,179.236,19.380,152.347
C05382=1099.343,365.876,-89.921,179.233,19.376,152.347
C05383=1099.337,365.629,-89.886,179.230,19.372,152.347
C05384=1099.332,365.381,-89.851,179.227,19.367,152.346
C05385=1099.326,365.134,-89.816,179.225,19.363,152.345
C05386=1099.320,364.886,-89.780,179.222,19.359,152.345
C05387=1099.315,364.639,-89.745,179.218,19.354,152.344
C05388=1099.308,364.392,-89.710,179.215,19.350,152.344
C05389=1099.303,364.144,-89.675,179.213,19.346,152.343
C05390=1099.297,363.896,-89.639,179.210,19.342,152.343
C05391=1099.291,363.649,-89.604,179.206,19.337,152.342
C05392=1099.286,363.402,-89.568,179.204,19.333,152.342
C05393=1099.280,363.154,-89.533,179.201,19.329,152.341
C05394=1099.274,362.908,-89.499,179.198,19.325,152.341
C05395=1099.268,362.660,-89.463,179.195,19.321,152.341
C05396=1099.263,362.413,-89.428,179.192,19.316,152.340
C05397=1099.257,362.165,-89.393,179.189,19.312,152.340
C05398=1099.251,361.918,-89.357,179.186,19.308,152.339
C05399=1099.245,361.670,-89.323,179.183,19.304,152.339
C05400=1099.240,361.423,-89.287,179.180,19.300,152.338
C05401=1099.234,361.176,-89.252,179.177,19.295,152.338
C05402=1099.228,360.927,-89.217,179.174,19.291,152.337
C05403=1099.222,360.681,-89.182,179.171,19.287,152.337
C05404=1099.216,360.432,-89.147,179.168,19.283,152.336
C05405=1099.211,360.185,-89.112,179.165,19.279,152.336
C05406=1099.206,359.938,-89.077,179.162,19.275,152.335
C05407=1099.199,359.690,-89.042,179.159,19.271,152.335
C05408=1099.194,359.443,-89.007,179.156,19.267,152.335
C05409=1099.187,359.196,-88.972,179.153,19.263,152.334
C05410=1099.182,358.948,-88.938,179.150,19.259,152.334
C05411=1099.177,358.701,-88.902,179.147,19.255,152.333
C05412=1099.170,358.453,-88.868,179.144,19.251,152.333
C05413=1099.165,358.205,-88.833,179.141,19.247,152.332
C05414=1099.160,357.958,-88.798,179.138,19.243,152.332
C05415=1099.153,357.710,-88.763,179.135,19.239,152.332
C05416=1099.148,357.463,-88.728,179.132,19.235,152.331
C05417=1099.139,357.086,-88.675,179.128,19.229,152.331
C05418=1099.131,356.710,-88.623,179.123,19.223,152.330
C05419=1099.121,356.333,-88.570,179.118,19.218,152.329
C05420=1099.112,355.957,-88.517,179.114,19.211,152.329
C05421=1099.107,355.709,-88.483,179.111,19.207,152.328
C05422=1099.101,355.462,-88.448,179.108,19.204,152.328
C05423=1099.096,355.215,-88.413,179.105,19.200,152.328
C05424=1099.090,354.967,-88.379,179.101,19.195,152.327
C05425=1099.084,354.719,-88.344,179.099,19.192,152.327
C05426=1099.079,354.472,-88.310,179.095,19.188,152.327
C05427=1099.073,354.223,-88.275,179.093,19.185,152.326
C05428=1099.067,353.977,-88.240,179.089,19.180,152.326
C05429=1099.062,353.729,-88.206,179.087,19.177,152.325
C05430=1099.056,353.482,-88.172,179.084,19.173,152.325
C05431=1099.050,353.234,-88.137,179.080,19.169,152.325
C05432=1099.044,352.986,-88.103,179.077,19.165,152.324
C05433=1099.038,352.739,-88.069,179.074,19.161,152.324
C05434=1099.033,352.492,-88.034,179.071,19.158,152.324
C05435=1099.027,352.244,-88.000,179.068,19.154,152.323
C05436=1099.022,351.996,-87.965,179.065,19.150,152.323
C05437=1099.016,351.749,-87.931,179.062,19.147,152.323
C05438=1099.010,351.501,-87.897,179.059,19.143,152.322
C05439=1099.004,351.253,-87.862,179.056,19.139,152.322
C05440=1098.998,351.006,-87.828,179.053,19.136,152.322
C05441=1098.992,350.758,-87.794,179.050,19.132,152.321
C05442=1098.987,350.511,-87.760,179.046,19.128,152.321
C05443=1098.982,350.263,-87.726,179.044,19.125,152.321
C05444=1098.975,350.015,-87.691,179.040,19.121,152.320
C05445=1098.969,349.768,-87.657,179.037,19.117,152.320
C05446=1098.964,349.520,-87.623,179.034,19.113,152.320
